# B&R Automation Studio project lab1_MIRTS_save2_4
Automation Studio 4.5.2.102

## Configuration Config1

### Task classes (Cpu.sw)
```
Cyclic#1:
  Program <- Program.prg
Cyclic#4:
  Program1 <- Program1.prg
Binaries: udbdef, TCData, ashwac, arconfig, asfw, ashwd, iomap, User, Role, sysconf
Libraries: MotorCntrl
```

## Configuration labBR

### IoMap.iom - 4PP065_0571_P74/IoMap.iom
```iecst
VAR_CONFIG
	::DoorCtrl:DoorBlock.sw1 AT %IX."X20DI9371".DigitalInput03;
	::DoorCtrl:DoorBlock.sw2 AT %IX."X20DI9371".DigitalInput04;
	::DoorCtrl:DoorBlock.sw3 AT %IX."X20DI9371".DigitalInput05;
	::DoorCtrl:CMD AT %QW."8I64xxxxxxx.00x-1".CMDD_Output;
	::DoorCtrl:ETAD AT %IW."8I64xxxxxxx.00x-1".ETAD_Input;
	::DoorCtrl:Speed AT %QW."8I64xxxxxxx.00x-1".LFRD_Output;
	::LedCtrl:sc0 AT %QX."X20DO9322".DigitalOutput02;
	::LedCtrl:sc1 AT %QX."X20DO9322".DigitalOutput03;
	::LedCtrl:sc2 AT %QX."X20DO9322".DigitalOutput04;
	::LedCtrl:sc3  AT %QX."X20DO9322".DigitalOutput05;
	::DoorCtrl:DoorBlock.sw0 AT %IX."X20DI9371".DigitalInput02;
	::DoorCtrl:DoorBlock.direction AT %IX."X20DI9371".DigitalInput01;
END_VAR
```

### Acp10map.ncm - 4PP065_0571_P74/Motion/Acp10map.ncm
```
NcMapping (NcSwId=Acp10)
  NcObject gAxis01 (ModuleId=X20SM1436, ModuleAddress=SDC_IF1.ST1, Type=ncAXIS, Channel=1, AcoposSimulation=Off, InitParameter=gAxis01i, AcoposParameter=gAxis01a, AdditionalData=CNC_Enabled="1" , Disabled=FALSE, ModuleDisabled=FALSE)
  NcObject gAxis02 (ModuleId=X20SM1436a, ModuleAddress=SDC_IF1.ST2, Type=ncAXIS, Channel=1, AcoposSimulation=Off, InitParameter=gAxis02i, AcoposParameter=gAxis02a, Disabled=FALSE, ModuleDisabled=FALSE)
  NcObject gAxis03 (ModuleId=8I64xxxxxxx.00x-1, ModuleAddress=SDC_IF1.ST3, Type=ncAXIS, Channel=1, AcoposSimulation=Off, InitParameter=gAxis03i, AcoposParameter=gAxis03a, AdditionalData=CNC_Enabled="1" , Disabled=FALSE, ModuleDisabled=FALSE)
  NcObject gAxis04 (ModuleId=X20SM1436b, ModuleAddress=SDC_IF1.ST4, Type=ncAXIS, Channel=1, AcoposSimulation=Off, InitParameter=gAxis04i, AcoposParameter=gAxis04a, AdditionalData=CNC_Enabled="1" , Disabled=FALSE, ModuleDisabled=FALSE)
  NcObject gAxis05 (ModuleId=X20SM1436c, ModuleAddress=SDC_IF1.ST5, Type=ncAXIS, Channel=1, AcoposSimulation=Off, InitParameter=gAxis05i, AcoposParameter=gAxis05a, Disabled=FALSE, ModuleDisabled=FALSE)
```

## Logical view

Binary libraries used (declarations not repeated): Runtime, Operator, AsIecCon, astime, sys_lib, asstring

### Global.var - Global variables
```iecst
VAR
	sw1 : BOOL := FALSE;
	sw2 : BOOL := FALSE;
	sw3 : BOOL := FALSE;
	sw0 : BOOL := FALSE;
END_VAR
```

### Package Logical/Libraries - Global libraries

- Library Logical/Libraries/X64Lib (ANSIC) (no source held here)

### Library Logical/Libraries/GateCtrl (ANSIC)

#### Types.typ
```iecst
TYPE
	GateState :
		(
		ST_INIT := 0,
		ST_UNKNOWN := 1,
		ST_OPEN := 2,
		ST_CLOSE := 3,
		ST_ACC_POS := 4,
		ST_ACC_NEG := 5,
		ST_POS := 6,
		ST_NEG := 7,
		ST_DEC_POS := 8,
		ST_DEC_NEG := 9
		);
END_TYPE
```

#### GateCtrl.fun
```iecst
FUNCTION_BLOCK FBLed
	VAR_OUTPUT
		s1 : BOOL;
		s2 : BOOL;
		s3 : BOOL;
		s4 : BOOL;
	END_VAR
	VAR_INPUT
		State : {REDUND_UNREPLICABLE} GateState;
	END_VAR
END_FUNCTION_BLOCK

{REDUND_ERROR} FUNCTION_BLOCK FBGate (* *) (*$GROUP=User,$CAT=User,$GROUPICON=User.png,$CATICON=User.png*)
	VAR_INPUT
		sw0 : BOOL; (*инпут датчиков*)
		sw1 : BOOL;
		sw2 : BOOL;
		sw3 : BOOL;
		State : {REDUND_UNREPLICABLE} GateState;
		direction : BOOL;
	END_VAR
	VAR_OUTPUT
		Speed : INT;
	END_VAR
	VAR
		DriveBlk : FBX64Inverter;
	END_VAR
END_FUNCTION_BLOCK
```

#### FBGate.c
```c
#include <bur/plctypes.h>
#ifdef __cplusplus
	extern "C"
	{
#endif
	#include "GateCtrl.h"
#ifdef __cplusplus
	};
#endif
/* TODO: Add your comment here */
void FBGate(struct FBGate* inst)
{
	switch (inst->State) {
		case ST_INIT: //
			inst->State = ST_UNKNOWN;
			break;
		case ST_UNKNOWN: //
			if ((inst->direction == 0) && (inst->sw0 == 0)){
			inst->State = ST_OPEN;
			}
			if ((inst->direction == 1) && (inst->sw0 == 1)){
				inst->State = ST_CLOSE;
			}
			break;
		case ST_OPEN: //
			inst->DriveBlk.enable = 0;
			FBX64Inverter(&inst->DriveBlk);
			inst->Speed = 0;
			FBX64Inverter(&inst->DriveBlk);
			if (inst->direction == 1){
				inst->State = ST_ACC_POS;
			}
			break;
		case ST_CLOSE:
			inst->DriveBlk.enable = 0;
			FBX64Inverter(&inst->DriveBlk);
			inst->Speed = 0;
			FBX64Inverter(&inst->DriveBlk);
			if (inst->direction == 0){
				inst->State = ST_ACC_NEG;
			}
			break;
		case ST_ACC_POS:
			inst->DriveBlk.enable = 1;
			inst->Speed = 100;
			FBX64Inverter(&inst->DriveBlk);
			if (inst->sw1){
				inst->State = ST_POS;
			}
			if (inst->direction == 0) {
				inst->State = ST_ACC_NEG;
			}
			break;
		case ST_ACC_NEG:
			inst->DriveBlk.enable = 1;
			FBX64Inverter(&inst->DriveBlk);
			inst->Speed = -100;
			if (!inst->sw2){
				inst->State = ST_NEG;
			}
			break;
		case ST_NEG:
			inst->Speed = -300;
			FBX64Inverter(&inst->DriveBlk);
			if (!inst->sw1){
				inst->State = ST_DEC_NEG;
			}
			break;
		case ST_DEC_NEG:
			inst->Speed = -100;
			FBX64Inverter(&inst->DriveBlk);
			if (!inst->sw0){
				inst->State = ST_OPEN;
			}
			break;
		case ST_DEC_POS:
			FBX64Inverter(&inst->DriveBlk);
			inst->Speed = 100;
			if (inst->sw3){
				inst->State = ST_CLOSE;
			}
			break;
		case ST_POS:
			FBX64Inverter(&inst->DriveBlk);
			inst->Speed = 300;
			if (inst->sw2){
				inst->State = ST_DEC_POS;
			}
			if (inst->direction == 0) {
				inst->State = ST_NEG;
			}
			break;
	}
}
```

### arnc0man.typ
```iecst
TYPE
ARNC0SWVER_typ : STRUCT                                     (* Software Version ID *)
   NOT_USE_1            : ARRAY [0..1] OF USINT ;
   nc_system_device     : UINT ;                            (* ACOPOS operating system *)
   nc_manager           : UINT ;                            (* NC manager *)
   nc_system            : UINT ;                            (* NC operating system *)
END_STRUCT;
ARNC0OBIHW_typ : STRUCT                                     (* Hardware information *)
   init                 : USINT ;                           (* Initialized *)
   reserve1             : USINT ;                           (* Reserved *)
   acp_id               : USINT ;                           (* ACOPOS ID *)
   acp_id_nr            : USINT ;                           (* ACOPOS ID production number *)
   acp_typ              : USINT ;                           (* ACOPOS type *)
   ax_num               : USINT ;                           (* Number of axes (power stages) *)
   reserve2             : UINT ;                            (* Reserved *)
   product_code         : UDINT ;                           (* Product code *)
   serial_nr            : UDINT ;                           (* Serial number *)
END_STRUCT;
ARNC0OBINF_typ : STRUCT                                     (* NC Object Information *)
   net_if_typ           : UINT ;                            (* Network interface type *)
   net_if_idx           : UINT ;                            (* Network interface index *)
   node_nr              : UINT ;                            (* Drive node number *)
   nc_obj_typ           : UINT ;                            (* NC object type *)
   nc_obj_idx           : UINT ;                            (* NC object index *)
   reserve              : UINT ;                            (* Reserved *)
   nc_obj_name          : ARRAY [0..47] OF USINT ;          (* NC object name *)
   hardware             : ARNC0OBIHW_typ ;                  (* Hardware information *)
END_STRUCT;
ARNC0AXSIM_typ : STRUCT                                     (* Simulation mode *)
   NOT_USE_1            : ARRAY [0..3] OF USINT ;
   status               : UINT ;                            (* Status *)
   mode                 : UINT ;                            (* Mode *)
   NOT_USE_2            : ARRAY [0..47] OF USINT ;
END_STRUCT;
ARNC0GLIPA_typ : STRUCT                                     (* INIT Parameters *)
   ok                   : USINT ;                           (* Operation complete *)
   error                : USINT ;                           (* Error *)
   reserve              : UINT ;                            (* Reserved *)
   datobj_ident         : UDINT ;                           (* Data object ident *)
   data_modul           : ARRAY [0..11] OF USINT ;          (* Name of the data module *)
END_STRUCT;
ARNC0GLINI_typ : STRUCT                                     (* Global Initialization *)
   init                 : USINT ;                           (* Global Initialization complete *)
   NOT_USE_1            : ARRAY [0..2] OF USINT ;
   init_par             : ARNC0GLIPA_typ ;                  (* INIT Parameters *)
END_STRUCT;
ARNC0NSVRQ_typ : STRUCT                                     (* Request (to the drive) *)
   par_id               : UINT ;                            (* Parameter ID *)
   NOT_USE_1            : ARRAY [0..1] OF USINT ;
END_STRUCT;
ARNC0NSVRS_typ : STRUCT                                     (* Response (from the drive) *)
   par_id               : UINT ;                            (* Parameter ID *)
   NOT_USE_1            : ARRAY [0..1] OF USINT ;
END_STRUCT;
ARNC0NETSV_typ : STRUCT                                     (* Service Interface *)
   data_adr             : UDINT ;                           (* Data address *)
   data_text            : ARRAY [0..31] OF USINT ;          (* Data in text format *)
   request              : ARNC0NSVRQ_typ ;                  (* Request (to the drive) *)
   response             : ARNC0NSVRS_typ ;                  (* Response (from the drive) *)
END_STRUCT;
ARNC0NETAX_typ : STRUCT                                     (* Network *)
   init                 : USINT ;                           (* Network initialized *)
   phase                : USINT ;                           (* Phase *)
   NOT_USE_1            : USINT ;
   nc_sys_restart       : USINT ;                           (* A Restart of the NC operating system was executed *)
   reserve              : UINT ;                            (* Reserved *)
   reserve1             : UINT ;                            (* Reserved *)
   service              : ARNC0NETSV_typ ;                  (* Service Interface *)
END_STRUCT;
ARNC0AXDBS_typ : STRUCT                                     (* Status *)
   ok                   : USINT ;                           (* Operation complete *)
   error                : USINT ;                           (* Error *)
   reserve1             : USINT ;                           (* Reserved *)
   reserve2             : USINT ;                           (* Reserved *)
   data_len             : UDINT ;                           (* Length of data *)
   datobj_ident         : UDINT ;                           (* Data object ident *)
   datobj_datadr        : UDINT ;                           (* Address of the data object data *)
END_STRUCT;
ARNC0AXDBP_typ : STRUCT                                     (* Parameters *)
   file_device          : ARRAY [0..31] OF USINT ;          (* Name of File Device *)
   datobj_name          : ARRAY [0..31] OF USINT ;          (* Name of the data object *)
   datobj_type          : UINT ;                            (* Type of the data object *)
   datblock_par_id      : UINT ;                            (* Parameter ID of the data block *)
   idx1_par_id          : UINT ;                            (* Parameter ID of data block index 1 *)
   idx1                 : UINT ;                            (* Data block index 1 *)
   idx2_par_id          : UINT ;                            (* Parameter ID of data block index 2 *)
   idx2                 : UINT ;                            (* Data block index 2 *)
   NOT_USE_1            : ARRAY [0..7] OF USINT ;
END_STRUCT;
ARNC0AXDBL_typ : STRUCT                                     (* Data block operation *)
   status               : ARNC0AXDBS_typ ;                  (* Status *)
   parameter            : ARNC0AXDBP_typ ;                  (* Parameters *)
END_STRUCT;
ARNC0DISTA_typ : STRUCT                                     (* Status *)
   reference            : USINT ;                           (* Reference switch *)
   pos_hw_end           : USINT ;                           (* Positive HW end switch *)
   neg_hw_end           : USINT ;                           (* Negative HW end switch *)
   trigger1             : USINT ;                           (* Trigger1 *)
   trigger2             : USINT ;                           (* Trigger2 *)
   enable               : USINT ;                           (* Enable *)
   NOT_USE_1            : ARRAY [0..1] OF USINT ;
END_STRUCT;
ARNC0DILEV_typ : STRUCT                                     (* Active Input Level *)
   reference            : UINT ;                            (* Reference switch *)
   pos_hw_end           : UINT ;                            (* Positive HW end switch *)
   neg_hw_end           : UINT ;                            (* Negative HW end switch *)
   trigger1             : UINT ;                            (* Trigger1 *)
   trigger2             : UINT ;                            (* Trigger2 *)
   NOT_USE_1            : ARRAY [0..1] OF USINT ;
END_STRUCT;
ARNC0DIFRC_typ : STRUCT                                     (* Set status of digital inputs via force function *)
   reference            : USINT ;                           (* Reference switch *)
   pos_hw_end           : USINT ;                           (* Positive HW end switch *)
   neg_hw_end           : USINT ;                           (* Negative HW end switch *)
   trigger1             : USINT ;                           (* Trigger1 *)
   trigger2             : USINT ;                           (* Trigger2 *)
   reserve1             : USINT ;                           (* Reserved *)
   reserve2             : UINT ;                            (* Reserved *)
END_STRUCT;
ARNC0DIGIN_typ : STRUCT                                     (* Digital Inputs *)
   init                 : USINT ;                           (* Digital inputs initialized *)
   NOT_USE_1            : ARRAY [0..2] OF USINT ;
   status               : ARNC0DISTA_typ ;                  (* Status *)
   level                : ARNC0DILEV_typ ;                  (* Active Input Level *)
   force                : ARNC0DIFRC_typ ;                  (* Set status of digital inputs via force function *)
END_STRUCT;
ARNC0ENCSL_typ : STRUCT                                     (* Load *)
   units                : UDINT ;                           (* Units at the load *)
   rev_motor            : UDINT ;                           (* Motor revolutions *)
END_STRUCT;
ARNC0ENCSC_typ : STRUCT                                     (* Scale of encoder interface *)
   load                 : ARNC0ENCSL_typ ;                  (* Load *)
END_STRUCT;
ARNC0ENCPA_typ : STRUCT                                     (* Parameters of encoder interface *)
   count_dir            : USINT ;                           (* Count direction *)
   NOT_USE_1            : ARRAY [0..2] OF USINT ;
   scaling              : ARNC0ENCSC_typ ;                  (* Scaling *)
END_STRUCT;
ARNC0ENCIF_typ : STRUCT                                     (* Encoder interface *)
   init                 : USINT ;                           (* Encoder interface initialized *)
   NOT_USE_1            : ARRAY [0..2] OF USINT ;
   parameter            : ARNC0ENCPA_typ ;                  (* Parameters *)
END_STRUCT;
ARNC0AXLPA_typ : STRUCT                                     (* Parameters *)
   v_pos                : REAL ;                            (* Speed in positive direction *)
   v_neg                : REAL ;                            (* Speed in negative direction *)
   a1_pos               : REAL ;                            (* Acceleration in positive direction *)
   a2_pos               : REAL ;                            (* Deceleration in positive direction *)
   a1_neg               : REAL ;                            (* Acceleration in negative direction *)
   a2_neg               : REAL ;                            (* Deceleration in negative direction *)
   t_jolt               : REAL ;                            (* Jolt time *)
   t_in_pos             : REAL ;                            (* Settling time before message "In Position" *)
   pos_sw_end           : DINT ;                            (* Positive SW end *)
   neg_sw_end           : DINT ;                            (* Negative SW end *)
   sw_end_enable        : USINT ;                           (* Control byte for limit monitor *)
   sl_chain             : USINT ;                           (* Slaves in a chain or ncOFF *)
   NOT_USE_1            : ARRAY [0..1] OF USINT ;
   ds_warning           : REAL ;                            (* Lag error limit for display of a warning *)
   ds_stop              : REAL ;                            (* Lag error limit for stop of a movement *)
   a_stop               : REAL ;                            (* Acceleration limit for stop of a movement *)
   dv_stop              : REAL ;                            (* Speed error limit for stop of a movement *)
   dv_stop_mode         : UDINT ;                           (* Mode for speed error monitoring *)
END_STRUCT;
ARNC0AXLIM_typ : STRUCT                                     (* Limit values *)
   init                 : USINT ;                           (* Axis limit values initialized *)
   status               : USINT ;                           (* Status *)
   NOT_USE_1            : ARRAY [0..1] OF USINT ;
   parameter            : ARNC0AXLPA_typ ;                  (* Parameters *)
END_STRUCT;
ARNC0CTRPO_typ : STRUCT                                     (* Position controller *)
   kv                   : REAL ;                            (* Proportional amplification *)
   tn                   : REAL ;                            (* Integral action time *)
   t_predict            : REAL ;                            (* Prediction time *)
   t_total              : REAL ;                            (* Total time *)
   p_max                : REAL ;                            (* Maximum proportional action *)
   i_max                : REAL ;                            (* Maximum integral action *)
END_STRUCT;
ARNC0ISQFI_typ : STRUCT                                     (* ISQ Filter *)
   type                 : UINT ;                            (* Type *)
   reserve              : UINT ;                            (* Reserved *)
   a0                   : REAL ;                            (* Coefficient a0 *)
   a1                   : REAL ;                            (* Coefficient a1 *)
   b0                   : REAL ;                            (* Coefficient b0 *)
   b1                   : REAL ;                            (* Coefficient b1 *)
   b2                   : REAL ;                            (* Coefficient b2 *)
   c0_par_id            : UINT ;                            (* Parameter ID for coefficient c0 *)
   c1_par_id            : UINT ;                            (* Parameter ID for coefficient c1 *)
END_STRUCT;
ARNC0CTRSP_typ : STRUCT                                     (* Speed controller *)
   kv                   : REAL ;                            (* Proportional amplification *)
   tn                   : REAL ;                            (* Integral action time *)
   t_filter             : REAL ;                            (* Filter time constant *)
   isq_filter1          : ARNC0ISQFI_typ ;                  (* ISQ Filter1 *)
   isq_filter2          : ARNC0ISQFI_typ ;                  (* ISQ Filter2 *)
   isq_filter3          : ARNC0ISQFI_typ ;                  (* ISQ Filter3 *)
END_STRUCT;
ARNC0CTRUF_typ : STRUCT                                     (* U/f Control *)
   type                 : USINT ;                           (* Type *)
   auto_config          : USINT ;                           (* Automatic configuration *)
   reserve              : UINT ;                            (* Reserved *)
   u0                   : REAL ;                            (* Boost voltage *)
   un                   : REAL ;                            (* Rated voltage *)
   fn                   : REAL ;                            (* Rated frequency *)
   k_f_slip             : REAL ;                            (* Slip compensation: Multiplication factor of compensated frequency *)
END_STRUCT;
ARNC0CTRFF_typ : STRUCT                                     (* Feed Forward Control *)
   torque_load          : REAL ;                            (* Load torque *)
   torque_pos           : REAL ;                            (* Torque in positive direction *)
   torque_neg           : REAL ;                            (* Torque in negative direction *)
   kv_torque            : REAL ;                            (* Speed torque factor *)
   inertia              : REAL ;                            (* Mass moment of inertia *)
   t_filter_a           : REAL ;                            (* Acceleration filter time constant *)
END_STRUCT;
ARNC0CTRL_typ : STRUCT                                      (* Controller *)
   init                 : USINT ;                           (* Controller initialized *)
   ready                : USINT ;                           (* Ready *)
   status               : USINT ;                           (* Status *)
   mode                 : USINT ;                           (* Mode *)
   position             : ARNC0CTRPO_typ ;                  (* Position Controller *)
   speed                : ARNC0CTRSP_typ ;                  (* Speed Controller *)
   uf                   : ARNC0CTRUF_typ ;                  (* U/f Control *)
   ff                   : ARNC0CTRFF_typ ;                  (* Feed Forward Control *)
END_STRUCT;
ARNC0AXSTI_typ : STRUCT                                     (* Index of Parameter Record *)
   command              : USINT ;                           (* for the next stop command *)
   NOT_USE_1            : ARRAY [0..2] OF USINT ;
END_STRUCT;
ARNC0AXSTP_typ : STRUCT                                     (* Parameter Records *)
   decel_ramp           : USINT ;                           (* Deceleration ramp *)
   controller           : USINT ;                           (* Controller state after movement abortion *)
   NOT_USE_1            : ARRAY [0..1] OF USINT ;
END_STRUCT;
ARNC0AXSTQ_typ : STRUCT                                     (* Quickstop *)
   decel_ramp           : USINT ;                           (* Deceleration ramp *)
   NOT_USE_1            : USINT ;
   reserve2             : UINT ;                            (* Reserved *)
   NOT_USE_2            : ARRAY [0..3] OF USINT ;
END_STRUCT;
ARNC0AXSTD_typ : STRUCT                                     (* Drive error *)
   decel_ramp           : USINT ;                           (* Deceleration ramp *)
   reserve1             : USINT ;                           (* Reserved *)
   reserve2             : UINT ;                            (* Reserved *)
END_STRUCT;
ARNC0AXSTO_typ : STRUCT                                     (* Stop Movement *)
   init                 : USINT ;                           (* Stop initialized *)
   NOT_USE_1            : ARRAY [0..2] OF USINT ;
   index                : ARNC0AXSTI_typ ;                  (* Index *)
   parameter            : ARRAY [0..3] OF ARNC0AXSTP_typ ;  (* Parameter record *)
   quickstop            : ARNC0AXSTQ_typ ;                  (* Quickstop *)
   drive_error          : ARNC0AXSTD_typ ;                  (* Drive error *)
END_STRUCT;
ARNC0HOMST_typ : STRUCT                                     (* Status *)
   ok                   : USINT ;                           (* Reference position valid *)
   NOT_USE_1            : ARRAY [0..2] OF USINT ;
   tr_s_rel             : REAL ;                            (* Distance between activation of "triggering reference pulse" and the occurrence of the reference pulse *)
   offset               : DINT ;                            (* Home offset after completion of homing procedure *)
END_STRUCT;
ARNC0HOMPA_typ : STRUCT                                     (* Parameters *)
   s                    : DINT ;                            (* Reference position *)
   v_switch             : REAL ;                            (* Speed for searching the reference switch *)
   v_trigger            : REAL ;                            (* Trigger speed (after ref. switch has been reached) *)
   a                    : REAL ;                            (* Acceleration *)
   mode                 : USINT ;                           (* Mode *)
   edge                 : USINT ;                           (* Edge of reference switch *)
   start_dir            : USINT ;                           (* Start direction *)
   trigg_dir            : USINT ;                           (* Trigger direction *)
   ref_pulse            : USINT ;                           (* Reference pulse *)
   fix_dir              : USINT ;                           (* Fixed direction *)
   reserve1             : USINT ;                           (* Reserved *)
   reserve2             : USINT ;                           (* Reserved *)
   tr_s_block           : REAL ;                            (* Reference pulse block distance *)
   torque_lim           : REAL ;                            (* Torque limit for homing on block *)
   ds_block             : REAL ;                            (* Lag error for block detection *)
   ds_stop              : REAL ;                            (* Lag error for stop of a movement *)
END_STRUCT;
ARNC0HOME_typ : STRUCT                                      (* Homing *)
   init                 : USINT ;                           (* Homing procedure initialized *)
   NOT_USE_1            : ARRAY [0..2] OF USINT ;
   status               : ARNC0HOMST_typ ;                  (* Status *)
   parameter            : ARNC0HOMPA_typ ;                  (* Parameters *)
END_STRUCT;
ARNC0BMVST_typ : STRUCT                                     (* Status *)
   in_pos               : USINT ;                           (* "In Position" (target position reached) *)
   reserve              : ARRAY [0..2] OF USINT ;           (* Reserved *)
END_STRUCT;
ARNC0BMVOV_typ : STRUCT                                     (* Override *)
   v                    : UINT ;                            (* Speed override *)
   NOT_USE_1            : ARRAY [0..1] OF USINT ;
END_STRUCT;
ARNC0BMVPA_typ : STRUCT                                     (* Parameters *)
   s                    : DINT ;                            (* Target position or relative move distance *)
   v_pos                : REAL ;                            (* Speed in positive direction *)
   v_neg                : REAL ;                            (* Speed in negative direction *)
   a1_pos               : REAL ;                            (* Acceleration in positive direction *)
   a2_pos               : REAL ;                            (* Deceleration in positive direction *)
   a1_neg               : REAL ;                            (* Acceleration in negative direction *)
   a2_neg               : REAL ;                            (* Deceleration in negative direction *)
END_STRUCT;
ARNC0TRG_typ : STRUCT                                       (* Source for Hardware Trigger *)
   nc_object            : UDINT ;                           (* NC object or ncOFF *)
   NOT_USE_1            : ARRAY [0..7] OF USINT ;
END_STRUCT;
ARNC0TRSTP_typ : STRUCT                                     (* Mode "Stop after trigger" *)
   init                 : USINT ;                           (* Initialized *)
   event                : USINT ;                           (* Event *)
   NOT_USE_1            : ARRAY [0..1] OF USINT ;
   s_rest               : DINT ;                            (* Remaining distance after trigger *)
   trg_source           : ARNC0TRG_typ ;                    (* Trigger Source *)
END_STRUCT;
ARNC0BAMOV_typ : STRUCT                                     (* Basis Movements *)
   init                 : USINT ;                           (* Initialized *)
   reserve0             : ARRAY [0..2] OF USINT ;           (* Reserved *)
   status               : ARNC0BMVST_typ ;                  (* Status *)
   override             : ARNC0BMVOV_typ ;                  (* Override *)
   parameter            : ARNC0BMVPA_typ ;                  (* Parameters *)
   trg_stop             : ARNC0TRSTP_typ ;                  (* Mode "Stop after trigger" *)
END_STRUCT;
ARNC0AXMOV_typ : STRUCT                                     (* Axis Movement *)
   mode                 : UINT ;                            (* Mode *)
   detail               : UINT ;                            (* Detail *)
   stop                 : ARNC0AXSTO_typ ;                  (* Stop Movement *)
   homing               : ARNC0HOME_typ ;                   (* Homing procedure *)
   basis                : ARNC0BAMOV_typ ;                  (* Basis movements *)
END_STRUCT;
ARNC0SUOST_typ : STRUCT                                     (* Status *)
   ident                : UDINT ;                           (* Ident of data object *)
   ok                   : USINT ;                           (* Operation complete *)
   error                : USINT ;                           (* Error *)
   reserve1             : USINT ;                           (* Reserved *)
   reserve2             : USINT ;                           (* Reserved *)
END_STRUCT;
ARNC0SUOPA_typ : STRUCT                                     (* Parameters *)
   name                 : ARRAY [0..11] OF USINT ;          (* Name of data object *)
END_STRUCT;
ARNC0SUOBJ_typ : STRUCT                                     (* Data object *)
   status               : ARNC0SUOST_typ ;                  (* Status *)
   parameter            : ARNC0SUOPA_typ ;                  (* Parameters *)
END_STRUCT;
ARNC0SUMAS_typ : STRUCT                                     (* Status *)
   mode                 : UINT ;                            (* Mode *)
   ok                   : USINT ;                           (* Operation complete *)
   error                : USINT ;                           (* Error *)
   quality              : REAL ;                            (* Quality of parameter identification *)
END_STRUCT;
ARNC0SUMAO_typ : STRUCT                                     (* Optional parameters *)
   z_p                  : USINT ;                           (* Number of polepairs *)
   phase                : USINT ;                           (* Phase *)
   reserve2             : UINT ;                            (* Reserved *)
   u_const              : REAL ;                            (* Voltage constant *)
   v_max                : REAL ;                            (* Maximum speed *)
   trq_0                : REAL ;                            (* Stall  torque *)
   trq_n                : REAL ;                            (* Rated torque *)
   trq_max              : REAL ;                            (* Peak  torque *)
   trq_const            : REAL ;                            (* Torque constant *)
   i_0                  : REAL ;                            (* Stall current *)
   i_max                : REAL ;                            (* Peak current *)
   i_m                  : REAL ;                            (* Magnetizing current *)
   phase_cross_sect     : REAL ;                            (* Cross section of a phase *)
   invcl_a1             : REAL ;                            (* Inverter characteristic: Gain factor *)
   invcl_a2             : REAL ;                            (* Inverter characteristic: Exponent *)
END_STRUCT;
ARNC0SUMAP_typ : STRUCT                                     (* Parameters *)
   mode                 : UINT ;                            (* Mode *)
   reserve              : UINT ;                            (* Reserved *)
   u_n                  : REAL ;                            (* Rated voltage *)
   i_n                  : REAL ;                            (* Rated current *)
   v_n                  : REAL ;                            (* Rated speed *)
   f_n                  : REAL ;                            (* Rated frequency *)
   cos_phi              : REAL ;                            (* Active power factor *)
   t_tripping_therm     : REAL ;                            (* Tripping time at thermal overload *)
   optional             : ARNC0SUMAO_typ ;                  (* Optional parameters *)
END_STRUCT;
ARNC0SUMA_typ : STRUCT                                      (* Induction motor *)
   status               : ARNC0SUMAS_typ ;                  (* Status *)
   parameter            : ARNC0SUMAP_typ ;                  (* Parameters *)
END_STRUCT;
ARNC0SUMSS_typ : STRUCT                                     (* Status *)
   mode                 : UINT ;                            (* Mode *)
   ok                   : USINT ;                           (* Operation complete *)
   error                : USINT ;                           (* Error *)
   quality              : REAL ;                            (* Quality of parameter identification *)
END_STRUCT;
ARNC0SUMSO_typ : STRUCT                                     (* Optional parameters *)
   phase                : USINT ;                           (* Phase *)
   reserve1             : USINT ;                           (* Reserved *)
   reserve2             : UINT ;                            (* Reserved *)
   u_const              : REAL ;                            (* Voltage constant *)
   v_max                : REAL ;                            (* Maximum speed *)
   trq_0                : REAL ;                            (* Stall  torque *)
   trq_const            : REAL ;                            (* Torque constant *)
   i_0                  : REAL ;                            (* Stall current *)
   phase_cross_sect     : REAL ;                            (* Cross section of a phase *)
   invcl_a1             : REAL ;                            (* Inverter characteristic: Gain factor *)
   invcl_a2             : REAL ;                            (* Inverter characteristic: Exponent *)
END_STRUCT;
ARNC0SUMSP_typ : STRUCT                                     (* Parameters *)
   mode                 : UINT ;                            (* Mode *)
   z_p                  : USINT ;                           (* Number of polepairs *)
   reserve              : USINT ;                           (* Reserved *)
   u_n                  : REAL ;                            (* Rated voltage *)
   i_n                  : REAL ;                            (* Rated current *)
   v_n                  : REAL ;                            (* Rated speed *)
   trq_n                : REAL ;                            (* Rated torque *)
   trq_max              : REAL ;                            (* Peak  torque *)
   i_max                : REAL ;                            (* Peak current *)
   t_tripping_therm     : REAL ;                            (* Tripping time at thermal overload *)
   optional             : ARNC0SUMSO_typ ;                  (* Optional parameters *)
END_STRUCT;
ARNC0SUMS_typ : STRUCT                                      (* Synchronous motor *)
   status               : ARNC0SUMSS_typ ;                  (* Status *)
   parameter            : ARNC0SUMSP_typ ;                  (* Parameters *)
END_STRUCT;
ARNC0SUPHS_typ : STRUCT                                     (* Status *)
   mode                 : UINT ;                            (* Mode *)
   ok                   : USINT ;                           (* Operation complete *)
   error                : USINT ;                           (* Error *)
   rho_0                : REAL ;                            (* Commutation offset *)
   z_p                  : USINT ;                           (* Number of polepairs *)
   reserve1             : USINT ;                           (* Reserved *)
   reserve2             : UINT ;                            (* Reserved *)
END_STRUCT;
ARNC0SUPHP_typ : STRUCT                                     (* Parameters *)
   mode                 : UINT ;                            (* Mode *)
   reserve              : UINT ;                            (* Reserved *)
   i                    : REAL ;                            (* Current *)
   t                    : REAL ;                            (* Time *)
END_STRUCT;
ARNC0SUPH_typ : STRUCT                                      (* Motor phasing *)
   status               : ARNC0SUPHS_typ ;                  (* Status *)
   parameter            : ARNC0SUPHP_typ ;                  (* Parameters *)
END_STRUCT;
ARNC0SUCST_typ : STRUCT                                     (* Status *)
   mode                 : UINT ;                            (* Mode *)
   ok                   : USINT ;                           (* Operation complete *)
   error                : USINT ;                           (* Error *)
END_STRUCT;
ARNC0SUCPA_typ : STRUCT                                     (* Parameters *)
   mode                 : UINT ;                            (* Mode *)
   orientation          : USINT ;                           (* Orientation *)
   operating_point      : USINT ;                           (* Operating point *)
   i_max_percent        : REAL ;                            (* Maximum percentage for rated current *)
   v_max_percent        : REAL ;                            (* Maximum percentage for speed limit value *)
   s_max                : DINT ;                            (* Maximum move distance *)
   ds_max               : REAL ;                            (* Maximum lag error *)
   kv_percent           : REAL ;                            (* Percentage for proportional amplification *)
   signal_order         : UDINT ;                           (* Order of excitation signal *)
   kv_max               : REAL ;                            (* Maximum proportional amplification *)
   a                    : REAL ;                            (* Acceleration *)
   signal_type          : UINT ;                            (* Type of the excitation signal *)
   reserve              : UINT ;                            (* Reserved *)
   signal_f_start       : REAL ;                            (* Start frequency of the excitation signal *)
   signal_f_stop        : REAL ;                            (* Stop frequency of the excitation signal *)
   signal_time          : REAL ;                            (* Duration of the excitation signal *)
END_STRUCT;
ARNC0SUCTR_typ : STRUCT                                     (* Controller *)
   status               : ARNC0SUCST_typ ;                  (* Status *)
   parameter            : ARNC0SUCPA_typ ;                  (* Parameters *)
END_STRUCT;
ARNC0SUIRS_typ : STRUCT                                     (* Status *)
   mode                 : UINT ;                            (* Mode *)
   ok                   : USINT ;                           (* Operation complete *)
   error                : USINT ;                           (* Error *)
   quality              : REAL ;                            (* Quality of parameter identification *)
END_STRUCT;
ARNC0SUIRP_typ : STRUCT                                     (* Parameters *)
   mode                 : UINT ;                            (* Mode *)
   reserve              : USINT ;                           (* Reserved *)
   ref_system           : USINT ;                           (* Reference system *)
   pos_offset           : REAL ;                            (* Position offset *)
   v                    : REAL ;                            (* Speed *)
END_STRUCT;
ARNC0SUIR_typ : STRUCT                                      (* ISQ-Ripple *)
   status               : ARNC0SUIRS_typ ;                  (* Status *)
   parameter            : ARNC0SUIRP_typ ;                  (* Parameters *)
END_STRUCT;
ARNC0SETUP_typ : STRUCT                                     (* Setup *)
   status               : USINT ;                           (* Status *)
   reserve              : USINT ;                           (* Reserved *)
   detail               : UINT ;                            (* Detail *)
   datobj               : ARNC0SUOBJ_typ ;                  (* Data object *)
   motor_induction      : ARNC0SUMA_typ ;                   (* Induction motor *)
   motor_synchron       : ARNC0SUMS_typ ;                   (* Synchronous motor *)
   motor_phasing        : ARNC0SUPH_typ ;                   (* Motor phasing *)
   controller           : ARNC0SUCTR_typ ;                  (* Controller *)
   isq_ripple           : ARNC0SUIR_typ ;                   (* ISQ-Ripple *)
END_STRUCT;
ARNC0PLCOPENAX_typ : STRUCT                                 (* PLCopen *)
   PLCopen_AxState      : USINT ;                           (* PLCopen axis state *)
   NOT_USE_1            : ARRAY [0..2] OF USINT ;
END_STRUCT;
ARNC0ACTST_typ : STRUCT                                     (* Status *)
   active               : USINT ;                           (* Active *)
   complete             : USINT ;                           (* Complete *)
   NOT_USE_1            : ARRAY [0..1] OF USINT ;
END_STRUCT;
ARNC0LATCH_typ : STRUCT                                     (* Position latch *)
   status               : ARNC0ACTST_typ ;                  (* Status *)
   position             : DINT ;                            (* Latchposition *)
   position2            : DINT ;                            (* Second latchposition *)
   event                : USINT ;                           (* Event *)
   reserve              : ARRAY [0..2] OF USINT ;           (* Reserved *)
   window               : DINT ;                            (* Latch window *)
   w_position           : DINT ;                            (* Position of the latch window *)
END_STRUCT;
ARNC0POS_L_typ : STRUCT                                     (* Position latches *)
   latch1               : ARNC0LATCH_typ ;                  (* Positioning latch 1 *)
   latch2               : ARNC0LATCH_typ ;                  (* Positioning latch 2 *)
END_STRUCT;
ARNC0CPRST_typ : STRUCT                                     (* Status *)
   active               : USINT ;                           (* Active *)
   index                : USINT ;                           (* Index *)
   cnt_start            : USINT ;                           (* Number of not acknowledged start commands *)
   reserve              : USINT ;                           (* Reserved *)
   curr_prof            : ARRAY [0..11] OF USINT ;          (* Name of current cam profile *)
END_STRUCT;
ARNC0CPRPA_typ : STRUCT                                     (* Parameters *)
   mode                 : USINT ;                           (* Mode *)
   reserve0             : ARRAY [0..2] OF USINT ;           (* Reserved *)
   ma_ax                : UDINT ;                           (* NC object of the master axis *)
   ma_add_ax            : UDINT ;                           (* NC object of the additive axis of the master axis *)
   sl_add_ax            : UDINT ;                           (* NC object of the additive axis of the slave  axis *)
   ma_s_start           : DINT ;                            (* Start position of the master axis *)
   ma_ivstart           : UDINT ;                           (* Start interval of the master axis *)
   ma_add_el            : REAL ;                            (* "Additive" element of the master axis *)
   ma_factor            : REAL ;                            (* Multiplication factor for the master axis *)
   ma_add_fa            : REAL ;                            (* Multiplication factor for the "additive" axis of the master axis *)
   sl_add_el            : REAL ;                            (* "Additive" element of the slave axis *)
   sl_factor            : REAL ;                            (* Multiplication factor for the slave  axis *)
   sl_add_fa            : REAL ;                            (* Multiplication factor for the "additive" axis of the slave axis *)
   factor_set           : USINT ;                           (* Set multiplication factors "ma/sl_factor" *)
   reserve              : ARRAY [0..2] OF USINT ;           (* Reserved *)
   reserve1             : ARRAY [0..5] OF UDINT ;           (* Reserved *)
END_STRUCT;
ARNC0CPRDM_typ : STRUCT                                     (* Data Modules *)
   single               : ARRAY [0..11] OF USINT ;          (* Name of the entry cam profile *)
   cyclic               : ARRAY [0..11] OF USINT ;          (* Name of the cyclic cam profile *)
END_STRUCT;
ARNC0CPINF_typ : STRUCT                                     (* INFO Function *)
   status               : ARNC0ACTST_typ ;                  (* Status *)
   sl_s_rel             : DINT ;                            (* Relative position of slave axis in the cam profile *)
   ma_s_rel             : UDINT ;                           (* Relative position of master axis in the cam profile *)
END_STRUCT;
ARNC0CPRCG_typ : STRUCT                                     (* Compensation Gears *)
   ma_v_max             : REAL ;                            (* Maximum speed of the master axis *)
   ma_s_comp            : DINT ;                            (* Compensation distance of master axis *)
   sl_s_comp            : DINT ;                            (* Compensation distance of slave axis *)
END_STRUCT;
ARNC0CAMPR_typ : STRUCT                                     (* Electronic Cam Profile *)
   status               : ARNC0CPRST_typ ;                  (* Status *)
   parameter            : ARNC0CPRPA_typ ;                  (* Parameters *)
   data_modul           : ARNC0CPRDM_typ ;                  (* Data Modules *)
   info                 : ARNC0CPINF_typ ;                  (* INFO-function *)
   co_gears             : ARNC0CPRCG_typ ;                  (* Compensation gear *)
END_STRUCT;
ARNC0AUTSP_typ : STRUCT                                     (* Parameters *)
   index                : USINT ;                           (* Index *)
   reserve              : ARRAY [0..2] OF USINT ;           (* Reserved *)
END_STRUCT;
ARNC0AUTST_typ : STRUCT                                     (* Status *)
   init                 : USINT ;                           (* Initialized *)
   active               : USINT ;                           (* Active *)
   st_type              : USINT ;                           (* Type of the actual state *)
   st_index             : USINT ;                           (* Index of the actual state *)
   cam_prof             : ARNC0AUTSP_typ ;                  (* Cam profile *)
END_STRUCT;
ARNC0AUTID_typ : STRUCT                                     (* INIT State *)
   st_type              : USINT ;                           (* Type of the state to initialize *)
   st_index             : USINT ;                           (* Type of the state to initialize *)
   NOT_USE_1            : ARRAY [0..1] OF USINT ;
END_STRUCT;
ARNC0AUTCC_typ : STRUCT                                     (* Coupling Configuration *)
   ma_ax                : UDINT ;                           (* NC object of the master axis *)
   ma_add_ax            : UDINT ;                           (* NC object of the additive axis of the master axis *)
   sl_add_ax            : UDINT ;                           (* NC object of the additive axis of the slave  axis *)
END_STRUCT;
ARNC0AUTGL_typ : STRUCT                                     (* Global Parameters *)
   ma_add_el            : REAL ;                            (* "Additive" element of the master axis *)
   sl_add_el            : REAL ;                            (* "Additive" element of the slave axis *)
END_STRUCT;
ARNC0AUTEB_typ : STRUCT                                     (* Events for basis state *)
   type                 : USINT ;                           (* Type *)
   NOT_USE_1            : ARRAY [0..2] OF USINT ;
   trg_source           : ARNC0TRG_typ ;                    (* Trigger Source *)
   attribute            : USINT ;                           (* Attribute *)
   st_type              : USINT ;                           (* Type of the next state *)
   st_index             : USINT ;                           (* Index  of the next state *)
   NOT_USE_2            : USINT ;
END_STRUCT;
ARNC0AUTBA_typ : STRUCT                                     (* Basis State *)
   ma_s_start           : DINT ;                            (* Start position of the master axis *)
   ma_ivstart           : UDINT ;                           (* Start interval of the master axis *)
   event                : ARRAY [0..5] OF ARNC0AUTEB_typ ;  (* Event *)
END_STRUCT;
ARNC0AUTCG_typ : STRUCT                                     (* Compensation Gears *)
   ma_v_max             : REAL ;                            (* Maximum speed of the master axis *)
   ma_s_rel             : DINT ;                            (* Relative distance of the master axis *)
   sl_s_rel             : DINT ;                            (* Relative distance of the slave axis *)
   ma_s_min             : DINT ;                            (* Minimum distance of the master axis *)
   mode                 : USINT ;                           (* Mode *)
   reserve              : ARRAY [0..2] OF USINT ;           (* Reserved *)
END_STRUCT;
ARNC0AUTCP_typ : STRUCT                                     (* Cam Profile *)
   name                 : ARRAY [0..11] OF USINT ;          (* Name of the NC data module *)
   ma_factor            : REAL ;                            (* Multiplication factor for the master axis *)
   sl_factor            : REAL ;                            (* Multiplication factor for the slave  axis *)
END_STRUCT;
ARNC0AUTER_typ : STRUCT                                     (* Events for automat states *)
   type                 : USINT ;                           (* Type *)
   NOT_USE_1            : ARRAY [0..2] OF USINT ;
   trg_source           : ARNC0TRG_typ ;                    (* Trigger Source *)
   attribute            : USINT ;                           (* Attribute *)
   st_type              : USINT ;                           (* Type of the next state *)
   st_index             : USINT ;                           (* Index  of the next state *)
   NOT_USE_2            : USINT ;
END_STRUCT;
ARNC0AUTSC_typ : STRUCT                                     (* States *)
   count                : UINT ;                            (* Count *)
   NOT_USE_1            : ARRAY [0..1] OF USINT ;
   co_gears             : ARNC0AUTCG_typ ;                  (* Compensation gear *)
   cam_prof             : ARNC0AUTCP_typ ;                  (* Cam profile *)
   event                : ARRAY [0..5] OF ARNC0AUTER_typ ;  (* Event *)
END_STRUCT;
ARNC0AUTOM_typ : STRUCT                                     (* Cam Profile Automat *)
   status               : ARNC0AUTST_typ ;                  (* Status *)
   signal1              : USINT ;                           (* Signal 1 from the PLC to the cam profile automat *)
   signal2              : USINT ;                           (* Signal 2 from the PLC to the cam profile automat *)
   signal3              : USINT ;                           (* Signal 3 from the PLC to the cam profile automat *)
   signal4              : USINT ;                           (* Signal 4 from the PLC to the cam profile automat *)
   init_stat            : ARNC0AUTID_typ ;                  (* INIT State (for INIT of a certain state) *)
   coupling             : ARNC0AUTCC_typ ;                  (* Coupling configuration *)
   global               : ARNC0AUTGL_typ ;                  (* Global Parameters *)
   basis                : ARNC0AUTBA_typ ;                  (* Basis state *)
   state                : ARRAY [0..5] OF ARNC0AUTSC_typ ;  (* State *)
END_STRUCT;
ARNC0AXCMPST_typ : STRUCT                                   (* Status *)
   init                 : USINT ;                           (* Initialized *)
   mode                 : USINT ;                           (* Mode *)
   reserve0             : UINT ;                            (* Reserved *)
END_STRUCT;
ARNC0AXCMPSSE_typ : STRUCT                                  (* Slope error compensation *)
   data_modul1          : ARRAY [0..11] OF USINT ;          (* Name of data module 1 *)
   data_modul2          : ARRAY [0..11] OF USINT ;          (* Name of data module 2 *)
   set_factor           : REAL ;                            (* Multiplication factor for set values *)
   corr_factor          : REAL ;                            (* Multiplication factor for corrected values *)
   start_offset         : REAL ;                            (* Start offset *)
END_STRUCT;
ARNC0AXCMPBL_typ : STRUCT                                   (* Backlash compensation *)
   s_init               : REAL ;                            (* Initial relative movement to mesh *)
   s                    : REAL ;                            (* Backlash *)
   v                    : REAL ;                            (* Velocity *)
   a                    : REAL ;                            (* Acceleration *)
END_STRUCT;
ARNC0AXCMPPA_typ : STRUCT                                   (* Compensation parameter *)
   mode                 : USINT ;                           (* Mode *)
   reserve0             : ARRAY [0..2] OF USINT ;           (* Reserved *)
   slope                : ARNC0AXCMPSSE_typ ;               (* Slope error compensation *)
   backlash             : ARNC0AXCMPBL_typ ;                (* Backlash compensation *)
END_STRUCT;
ARNC0AXCMP_typ : STRUCT                                     (* Axis Compensation *)
   status               : ARNC0AXCMPST_typ ;                (* Status *)
   parameter            : ARNC0AXCMPPA_typ ;                (* Parameters *)
END_STRUCT;
ARNC0AXMOV2_typ : STRUCT                                    (* Extended Axis movement *)
   cam_prof             : ARNC0CAMPR_typ ;                  (* Cam profile *)
   automat              : ARNC0AUTOM_typ ;                  (* Cam profile automat *)
   compensation         : ARNC0AXCMP_typ ;                  (* Compensation of axis errors *)
END_STRUCT;
ARNC0AXMOS_typ : STRUCT                                     (* Status Bits *)
   ds_warning           : USINT ;                           (* Lag error greater than "limit.ds_warning" *)
   reserve              : ARRAY [0..2] OF USINT ;           (* Reserved *)
END_STRUCT;
ARNC0AXMON_typ : STRUCT                                     (* Axis monitor *)
   s_act                : DINT ;                            (* Actual position *)
   s_set                : DINT ;                            (* Set position *)
   s_set_comp           : REAL ;                            (* Compensated set position *)
   v_set                : REAL ;                            (* Set speed *)
   v_set_comp           : REAL ;                            (* Compensated set speed *)
   status               : ARNC0AXMOS_typ ;                  (* Status bits *)
   reserve0             : ARRAY [0..2] OF UDINT ;           (* Reserved *)
END_STRUCT;
ARNC0MSSTA_typ : STRUCT                                     (* Status *)
   err_cl0              : USINT ;                           (* Error class 0 *)
   NOT_USE_1            : ARRAY [0..2] OF USINT ;
END_STRUCT;
ARNC0MSCNT_typ : STRUCT                                     (* Number of not acknowledged messages *)
   error                : UINT ;                            (* Count of not acknowledged errors *)
   NOT_USE_1            : ARRAY [0..5] OF USINT ;
END_STRUCT;
ARNC0MSREC_typ : STRUCT                                     (* Current message record *)
   number               : UDINT ;                           (* Number *)
   info                 : ARRAY [0..11] OF USINT ;          (* Additional Info *)
   NOT_USE_1            : ARRAY [0..1] OF USINT ;
   errorclass           : UINT ;                            (* Error class *)
   reserve              : UDINT ;                           (* Reserved *)
END_STRUCT;
ARNC0MTXST_typ : STRUCT                                     (* Status of text determination *)
   lines                : UINT ;                            (* Lines of the determined text *)
   error                : UINT ;                            (* Error *)
END_STRUCT;
ARNC0MTXPA_typ : STRUCT                                     (* Parameters for text determination *)
   format               : UINT ;                            (* Format *)
   columns              : UINT ;                            (* Number of columns per line *)
   data_modul           : ARRAY [0..11] OF USINT ;          (* Name of the data module *)
   data_len             : UINT ;                            (* Length of data buffer in application program *)
   reserve              : UINT ;                            (* Reserved *)
   data_adr             : UDINT ;                           (* Address of data buffer in application program *)
END_STRUCT;
ARNC0MSTXT_typ : STRUCT                                     (* Text determination for current message record *)
   status               : ARNC0MTXST_typ ;                  (* Status *)
   parameter            : ARNC0MTXPA_typ ;                  (* Parameters *)
END_STRUCT;
ARNC0MSG_typ : STRUCT                                       (* Messages *)
   status               : ARNC0MSSTA_typ ;                  (* Status *)
   count                : ARNC0MSCNT_typ ;                  (* Count of not acknowledged messages *)
   record               : ARNC0MSREC_typ ;                  (* Current message record *)
   text                 : ARNC0MSTXT_typ ;                  (* Text determination for current message record *)
END_STRUCT;
ARNC0NCTST_typ : STRUCT                                     (* NC Test *)
   Open_UseApplNcObj    : USINT ;                           (* Open test: Use the same NC object as the application *)
   Close_NoMoveAbort    : USINT ;                           (* Close test: No move abortion *)
   reserve1             : USINT ;                           (* Reserved *)
   reserve2             : USINT ;                           (* Reserved *)
END_STRUCT;
ARNC0AXIS_typ : STRUCT                                      (* ARNC0 - Axis *)
   NOT_USE_1            : ARRAY [0..5] OF USINT ;
   size                 : UINT ;                            (* Size of the corresponding NC manager data type *)
   sw_version           : ARNC0SWVER_typ ;                  (* Software Version ID *)
   nc_obj_inf           : ARNC0OBINF_typ ;                  (* NC Object Information *)
   simulation           : ARNC0AXSIM_typ ;                  (* Simulation Mode *)
   global               : ARNC0GLINI_typ ;                  (* Global Parameters *)
   network              : ARNC0NETAX_typ ;                  (* Network *)
   datblock             : ARNC0AXDBL_typ ;                  (* Data block operation *)
   dig_in               : ARNC0DIGIN_typ ;                  (* Digital Inputs *)
   encoder_if           : ARNC0ENCIF_typ ;                  (* Encoder Interface *)
   limit                : ARNC0AXLIM_typ ;                  (* Limit value *)
   controller           : ARNC0CTRL_typ ;                   (* Controller *)
   move                 : ARNC0AXMOV_typ ;                  (* Axis movement *)
   setup                : ARNC0SETUP_typ ;                  (* Setup *)
   NOT_USE_2            : ARRAY [0..119] OF USINT ;
   PLCopen_MC           : ARNC0PLCOPENAX_typ ;              (* PLCopen for Motion Components *)
   pos_latch            : ARNC0POS_L_typ ;                  (* Positioning latch *)
   move2                : ARNC0AXMOV2_typ ;                 (* Extended axis movement *)
   monitor              : ARNC0AXMON_typ ;                  (* Monitor *)
   message              : ARNC0MSG_typ ;                    (* Messages (errors, warnings) *)
   nc_test              : ARNC0NCTST_typ ;                  (* NC Test *)
   NOT_USE_3            : ARRAY [0..47] OF USINT ;
END_STRUCT;
ARNC0CNCSIM_typ : STRUCT                                    (* Simulation mode *)
   status               : USINT ;                           (* Status *)
   reserve              : ARRAY [0..2] OF USINT ;           (* Reserved *)
END_STRUCT;
ARNC0ACCADEX_typ : STRUCT                                   (* Reference Address *)
   access_adr           : UDINT ;                           (* Address for "access" *)
END_STRUCT;
ARNC0NCLIM_typ : STRUCT                                     (* CNC limits *)
   init                 : USINT ;                           (* Initialization complete *)
   reserve              : ARRAY [0..2] OF USINT ;           (* Reserved *)
   v                    : REAL ;                            (* Velocity *)
   a_pos                : REAL ;                            (* Positive acceleration *)
   a_neg                : REAL ;                            (* Negative acceleration *)
   t_jolt               : REAL ;                            (* Jolt time *)
   blocktransition      : USINT ;                           (* Mode for block transitions *)
   reserve0             : ARRAY [0..2] OF USINT ;           (* Reserved *)
   v_jump               : REAL ;                            (* Speed jump *)
   a_jump               : REAL ;                            (* Acceleration jump *)
   v_jump_t             : REAL ;                            (* Speed jump for tangential axis *)
   s_jump_t             : REAL ;                            (* Tangential deviation for subsequent path elements *)
   s_sync1_t            : UINT ;                            (* Synchrone M-Function at end of path element *)
   s_sync2_t            : UINT ;                            (* Synchrone M-Function at beginn of path element *)
   radius_err           : REAL ;                            (* Error of radius *)
   block_buffer         : UDINT ;                           (* Block buffer for backtracing the CNC path *)
   elements             : UINT ;                            (* Calculated elements before starting *)
   lookahead            : UINT ;                            (* Size of lookahead buffer *)
   halt                 : USINT ;                           (* Stop at passing beyond the submission values *)
   reserve1             : ARRAY [0..2] OF USINT ;           (* Reserved *)
   filter_err           : REAL ;                            (* Maximum contour error caused by "axis[i],t_axfilter" *)
   filter_err_trans     : REAL ;                            (* Maximum contour error at block transition caused by "axis[i],t_axfilter" *)
   plot                 : ARNC0ACCADEX_typ ;                (* Plot buffer *)
   dynamic              : ARNC0ACCADEX_typ ;                (* Dynamic buffer *)
END_STRUCT;
ARNC0SKPLM_typ : STRUCT                                     (* Interpreter skip level *)
   level_0              : USINT ;                           (* Skip level 0 *)
   level_1              : USINT ;                           (* Skip level 1 *)
   level_2              : USINT ;                           (* Skip level 2 *)
   level_3              : USINT ;                           (* Skip level 3 *)
   level_4              : USINT ;                           (* Skip level 4 *)
   level_5              : USINT ;                           (* Skip level 5 *)
   level_6              : USINT ;                           (* Skip level 6 *)
   level_7              : USINT ;                           (* Skip level 7 *)
   level_8              : USINT ;                           (* Skip level 8 *)
   level_9              : USINT ;                           (* Skip level 9 *)
   reserve0             : ARRAY [0..1] OF USINT ;           (* Reserved *)
END_STRUCT;
ARNC0NCMST_typ : STRUCT                                     (* Status CNC movement *)
   cnt_ncprog           : UINT ;                            (* Number of started CNC programs/blocks *)
   halt                 : USINT ;                           (* State "halt" *)
   halt_info            : USINT ;                           (* INFO aboute cause of "Halt" state *)
   m1_stop              : USINT ;                           (* Operating mode "Stop at M1" *)
   single_s             : USINT ;                           (* Operating mode "Single step" *)
   skip_fcn             : USINT ;                           (* Operating mode "Skip Function" *)
   dpr_ovr              : USINT ;                           (* "normal" override \  DPR-override *)
   skip_level           : ARNC0SKPLM_typ ;                  (* Skip level *)
END_STRUCT;
ARNC0NCSTO_typ : STRUCT                                     (* Stop Movement *)
   decel_ramp           : USINT ;                           (* Deceleration ramp *)
   reserve0             : USINT ;                           (* Reserved *)
   reserve1             : UINT ;                            (* Reserved *)
END_STRUCT;
ARNC0NCESTO_typ : STRUCT                                    (* Emergency Stop *)
   path                 : USINT ;                           (* Path behaviour *)
   reserve0             : USINT ;                           (* Reserved *)
   reserve1             : UINT ;                            (* Reserved *)
END_STRUCT;
ARNC0NCPRG_typ : STRUCT                                     (* CNC program *)
   name                 : ARRAY [0..99] OF USINT ;          (* Name of the NC data module *)
   init_prg             : ARRAY [0..99] OF USINT ;          (* Name of initial CNC program *)
   start_pos_type       : USINT ;                           (* Type of start position *)
   start_mode           : USINT ;                           (* Start mode for CNC program *)
   NOT_USE_1            : USINT ;
   delete_mode          : USINT ;                           (* Mode for deleting a CNC program *)
   start_pos            : DINT ;                            (* Starting position *)
   restart_type         : USINT ;                           (* Type of restart point *)
   reserve1             : ARRAY [0..2] OF USINT ;           (* Reserved *)
   block_ncprog         : UDINT ;                           (* Block number in CNC program *)
   offset_ncprog        : UDINT ;                           (* Offset (Byte) in current CNC program *)
   s_ncprog             : REAL ;                            (* Path position in current CNC program *)
   s_start              : ARRAY [0..14] OF REAL ;           (* Starting position *)
END_STRUCT;
ARNC0ACCAD_typ : STRUCT                                     (* Address for evaluation with "access" *)
   access_adr           : UDINT ;                           (* Address for "access" *)
END_STRUCT;
ARNC0SSTEP_typ : STRUCT                                     (* Single step *)
   mode                 : USINT ;                           (* Mode *)
   reserve0             : ARRAY [0..2] OF USINT ;           (* Reserved *)
   bit_pattern          : UDINT ;                           (* Bit pattern *)
END_STRUCT;
ARNC0SKPL_typ : STRUCT                                      (* Interpreter skip level *)
   level_0              : USINT ;                           (* Skip level 0 *)
   level_1              : USINT ;                           (* Skip level 1 *)
   level_2              : USINT ;                           (* Skip level 2 *)
   level_3              : USINT ;                           (* Skip level 3 *)
   level_4              : USINT ;                           (* Skip level 4 *)
   level_5              : USINT ;                           (* Skip level 5 *)
   level_6              : USINT ;                           (* Skip level 6 *)
   level_7              : USINT ;                           (* Skip level 7 *)
   level_8              : USINT ;                           (* Skip level 8 *)
   level_9              : USINT ;                           (* Skip level 9 *)
   reserve0             : ARRAY [0..1] OF USINT ;           (* Reserved *)
END_STRUCT;
ARNC0NCMOV_typ : STRUCT                                     (* CNC movement *)
   status               : ARNC0NCMST_typ ;                  (* Status *)
   stop                 : ARNC0NCSTO_typ ;                  (* Stop Movement *)
   e_stop               : ARNC0NCESTO_typ ;                 (* Emergency stop *)
   override             : INT ;                             (* Override *)
   R_override           : UINT ;                            (* Rapid override affects CNC path *)
   F_override           : UDINT ;                           (* Feedrate override affects CNC path *)
   ncprogram            : ARNC0NCPRG_typ ;                  (* NC program *)
   ncblock              : ARRAY [0..51] OF USINT ;          (* NC block *)
   dpr_ovr              : ARNC0ACCAD_typ ;                  (* "normal" override \  DPR-override *)
   dpr_if               : ARNC0ACCAD_typ ;                  (* DPR-interface *)
   single_s             : ARNC0SSTEP_typ ;                  (* Operating mode "Single step" *)
   skip_level           : ARNC0SKPL_typ ;                   (* Skip level *)
END_STRUCT;
ARNC0NCDST_typ : STRUCT                                     (* CNC decoder status *)
   halt                 : USINT ;                           (* State "halt" *)
   sync                 : USINT ;                           (* State "Waiting for SYNC" *)
   breakpt_halt         : USINT ;                           (* State "Halt at breakpoint" *)
   single_s_halt        : USINT ;                           (* State "Halt in single step mode" *)
   single_s             : UINT ;                            (* Operating mode "Single step" *)
   reserve              : UINT ;                            (* Reserved *)
   program_load         : UINT ;                            (* Status of 'program load' *)
   program_unload       : UINT ;                            (* Status of 'program unload' *)
   mp_log               : USINT ;                           (* Motion packet log *)
   reserve1             : ARRAY [0..2] OF USINT ;           (* Reserved *)
END_STRUCT;
ARNC0DCHLTINFO_typ : STRUCT                                 (* Interpreter halt info (e.g. breakpoint, single step) *)
   file_name            : ARRAY [0..99] OF USINT ;          (* File name *)
   program_name         : ARRAY [0..99] OF USINT ;          (* Program name *)
   subprog_name         : ARRAY [0..99] OF USINT ;          (* Sub program name *)
   line_nr              : UDINT ;                           (* Line number *)
   block_nr             : UDINT ;                           (* Block number *)
END_STRUCT;
ARNC0DCCDC_typ : STRUCT                                     (* Cutting Diameter Correction *)
   side                 : USINT ;                           (* Processing side Cutting Diameter Compensation *)
   entry                : USINT ;                           (* Select/deselect Cutting Diameter Compensation *)
   circ_transition      : USINT ;                           (* Insert Circular Transitions *)
   circ_replace         : USINT ;                           (* Replace arc with straight line *)
   contour_violation    : USINT ;                           (* Accept contour violations *)
   intersection_path    : USINT ;                           (* Additional intersection path calculation *)
   NOT_USE_1            : ARRAY [0..1] OF USINT ;
   feedrate             : UDINT ;                           (* Feedrate on Transition Circles *)
   v_path_contour       : USINT ;                           (* Feedrate affects CNC path *)
   exit                 : USINT ;                           (* Deselection Mode Cutting Diameter Compensation *)
   NOT_USE_2            : ARRAY [0..1] OF USINT ;
END_STRUCT;
ARNC0DCPAR_typ : STRUCT                                     (* CNC decoder parameter *)
   move_cmd             : USINT ;                           (* Movement command *)
   plane                : USINT ;                           (* Plane *)
   co_ords              : USINT ;                           (* Co-ordinate definition *)
   center               : USINT ;                           (* Center point definition *)
   v_path               : UDINT ;                           (* Path speed *)
   cdc                  : ARNC0DCCDC_typ ;                  (* Tool radius correction *)
   t_ax_period          : USINT ;                           (* Operating mode for  tangential axis *)
   system_unit          : USINT ;                           (* Measurement unit for CNC system *)
   v_path_mode          : USINT ;                           (* Mode for feed rate calculation *)
   reserve1             : USINT ;                           (* Reserved *)
   rot_pref_dir         : USINT ;                           (* Preferable direction of rotary axes *)
   limit_switch_mode    : USINT ;                           (* Mode for axis limit switch *)
   reserve0             : ARRAY [0..1] OF USINT ;           (* Reserved *)
END_STRUCT;
ARNC0DCDMO_typ : STRUCT                                     (* CNC decoder datamodule *)
   status               : ARNC0ACTST_typ ;                  (* Status *)
   zero_tab             : ARRAY [0..11] OF USINT ;          (* Data module name of zero point offset table *)
   tool_tab             : ARRAY [0..11] OF USINT ;          (* Data module name of tool data table *)
   rpar_tab             : ARRAY [0..11] OF USINT ;          (* Data module name of R parameter  table *)
END_STRUCT;
ARNC0R_PAR_typ : STRUCT                                     (* CNC decorder R-parameters *)
   status               : ARNC0ACTST_typ ;                  (* Status *)
   index                : UINT ;                            (* Index *)
   NOT_USE_1            : ARRAY [0..1] OF USINT ;
   value                : REAL ;                            (* R-Parameter-Value *)
END_STRUCT;
ARNC0DCSST_typ : STRUCT                                     (* Step mode debugger *)
   mode                 : UINT ;                            (* Mode *)
   number               : UINT ;                            (* Number of blocks to halt after *)
END_STRUCT;
ARNC0DCBRKPT_typ : STRUCT                                   (* Set Breakpoint *)
   file_name            : ARRAY [0..99] OF USINT ;          (* File name *)
   program_name         : ARRAY [0..99] OF USINT ;          (* Program name *)
   block_nr             : UDINT ;                           (* Block number *)
   line_nr              : UDINT ;                           (* Line number *)
END_STRUCT;
ARNC0DCBRKINFO_typ : STRUCT                                 (* Breakpoint info *)
   total_nr             : UDINT ;                           (* Total number of currently set breakpoints *)
   breakpoint_set       : ARRAY [0..4] OF ARNC0DCBRKPT_typ ;  (* Info to currently set breakpoints *)
END_STRUCT;
ARNC0DCBRKPAR_typ : STRUCT                                  (* Breakpoint Parameter *)
   file_name            : ARRAY [0..99] OF USINT ;          (* File name *)
   pos_type             : UDINT ;                           (* Type of break point *)
   position             : UDINT ;                           (* Block or line number *)
   break_count          : UDINT ;                           (* Halt on n’th hit *)
END_STRUCT;
ARNC0DCBRK_typ : STRUCT                                     (* Breakpoint *)
   status               : ARNC0ACTST_typ ;                  (* Status *)
   info                 : ARNC0DCBRKINFO_typ ;              (* INFO-function *)
   parameter            : ARNC0DCBRKPAR_typ ;               (* Parameters *)
END_STRUCT;
ARNC0DCEXPR_typ : STRUCT                                    (* Expression *)
   status               : ARNC0ACTST_typ ;                  (* Status *)
   query                : ARRAY [0..63] OF USINT ;          (* Variable/expression to evaluate *)
   result               : ARRAY [0..63] OF USINT ;          (* Result *)
END_STRUCT;
ARNC0DCVACCINFO_typ : STRUCT                                (* Info for access to variables *)
   address              : UDINT ;                           (* Access address to interpreter variable *)
   length               : UDINT ;                           (* Variable size (total number of byte) *)
   array_dim1           : UDINT ;                           (* First array dimension *)
   array_dim2           : UDINT ;                           (* Second array dimension *)
   data_type            : UINT ;                            (* Data type (see AS library “sys_lib”) *)
   scope                : UINT ;                            (* Variable scope *)
   synch_type           : UINT ;                            (* Synchronization type *)
   reserve0             : UINT ;                            (* Reserved *)
END_STRUCT;
ARNC0RVARACC_typ : STRUCT                                   (* Access to variables *)
   status               : ARNC0ACTST_typ ;                  (* Status *)
   name                 : ARRAY [0..31] OF USINT ;          (* Name of variable *)
   info                 : ARNC0DCVACCINFO_typ ;             (* INFO-function *)
END_STRUCT;
ARNC0NCDEC_typ : STRUCT                                     (* CNC decoder *)
   init                 : USINT ;                           (* Initialization complete *)
   reserve              : ARRAY [0..2] OF USINT ;           (* Reserved *)
   status               : ARNC0NCDST_typ ;                  (* Status *)
   halt_info            : ARNC0DCHLTINFO_typ ;              (* INFO aboute cause of "Halt" state *)
   parameter            : ARNC0DCPAR_typ ;                  (* Parameters *)
   data_modul           : ARNC0DCDMO_typ ;                  (* Data Modules *)
   r_param              : ARNC0R_PAR_typ ;                  (* R-parameter *)
   s_step               : ARNC0DCSST_typ ;                  (* Interpreter single step mode *)
   breakpoint           : ARNC0DCBRK_typ ;                  (* Breakpoints in CNC program *)
   expression           : ARNC0DCEXPR_typ ;                 (* Variable/Expression watch and force function *)
   var_access           : ARNC0RVARACC_typ ;                (* Direct access to Interpreter Variables *)
END_STRUCT;
ARNC0NCAXST_typ : STRUCT                                    (* Status *)
   add_par_id           : UINT ;                            (* Parameter ID of the additive element for the cyclic set position *)
   reserve              : ARRAY [0..1] OF USINT ;           (* Reserved *)
END_STRUCT;
ARNC0TRC_typ : STRUCT                                       (* Trigger Configuration *)
   trigger1_pos         : USINT ;                           (* Trigger1: Positive edge *)
   trigger1_neg         : USINT ;                           (* Trigger1: Negative edge *)
   trigger2_pos         : USINT ;                           (* Trigger2: Positive edge *)
   trigger2_neg         : USINT ;                           (* Trigger2: Negative edge *)
END_STRUCT;
ARNC0NCTRG_typ : STRUCT                                     (* Source for Hardware Trigger *)
   nc_object            : UDINT ;                           (* NC object or ncOFF *)
   nc_object_plcopen    : UDINT ;                           (* NC object or ncOFF *)
   NOT_USE_1            : ARRAY [0..3] OF USINT ;
   trg_conf             : ARNC0TRC_typ ;                    (* Trigger Configuration *)
END_STRUCT;
ARNC0NCAXSSE_typ : STRUCT                                   (* Axes error compensation *)
   active               : USINT ;                           (* Active *)
   reserve              : ARRAY [0..2] OF USINT ;           (* Reserved *)
   cmp_data             : ARNC0ACCADEX_typ ;                (* Compensation data *)
END_STRUCT;
ARNC0NCAXP_typ : STRUCT                                     (* CNC-axis settings *)
   NOT_USE_1            : ARRAY [0..71] OF USINT ;
   status               : ARNC0NCAXST_typ ;                 (* Status *)
   nc_object            : UDINT ;                           (* NC object or ncOFF *)
   nc_object_plcopen    : UDINT ;                           (* NC object or ncOFF *)
   name                 : ARRAY [0..13] OF USINT ;          (* Name of the axis in the CNC program *)
   reserve3             : ARRAY [0..1] OF USINT ;           (* Reserved *)
   type                 : UDINT ;                           (* Type *)
   ipl_mode             : USINT ;                           (* Interpolation mode *)
   reserve4             : ARRAY [0..2] OF USINT ;           (* Reserved *)
   unitfactor           : REAL ;                            (* Multiplication factor of the units *)
   t_axfilter           : REAL ;                            (* Filter time for axis jolt filter *)
   drive_axfilter       : USINT ;                           (* Axis jolt filter on the drive during CNC movement *)
   reserve2             : ARRAY [0..2] OF USINT ;           (* Reserved *)
   rot_period           : REAL ;                            (* Period of rotary axis *)
   rot_offset           : REAL ;                            (* Start of period for rotary axis *)
   add_par_id           : UINT ;                            (* Parameter ID of the additive element for the cyclic set position *)
   reserve5             : ARRAY [0..1] OF USINT ;           (* Reserved *)
   trg_source           : ARNC0NCTRG_typ ;                  (* Trigger Source *)
   ax_compensation      : ARNC0NCAXSSE_typ ;                (* Axis error compensatioin *)
END_STRUCT;
ARNC0NCEXAXP_typ : STRUCT                                   (* External CNC axis parameters *)
   nc_object            : ARRAY [0..14] OF UDINT ;          (* NC object or ncOFF *)
END_STRUCT;
ARNC0NCAXCMP_typ : STRUCT                                   (* Compensation parameter for Cartesian axes *)
   matrix_el            : ARRAY [0..8] OF REAL ;            (* Element of compensation matrix *)
END_STRUCT;
ARNC0NCAXTRF_typ : STRUCT                                   (* Kinematic transformation parameters *)
   name                 : ARRAY [0..99] OF USINT ;          (* Name of the NC data module *)
   trf_full             : USINT ;                           (* Full kinematic transformation *)
   trf_type             : USINT ;                           (* Type of kinematic transformation *)
   reserve0             : ARRAY [0..1] OF USINT ;           (* Reserved *)
   axes_tcp             : ARRAY [0..11] OF USINT ;          (* Index of path axes *)
   axes_joint           : ARRAY [0..11] OF USINT ;          (* Index of joint axes *)
   axes_frame           : ARRAY [0..5] OF USINT ;           (* Index of frame axis [dx, dy, dz, phi, theta, psi] *)
   reserve1             : ARRAY [0..1] OF USINT ;           (* Reserved *)
   tcp_add_el           : ARRAY [0..11] OF REAL ;           (* Additive element of path axes *)
   joint_add_el         : ARRAY [0..11] OF REAL ;           (* Additive element of joint axes *)
   frame_add_el         : ARRAY [0..5] OF REAL ;            (* Additive element of frame axes *)
   d_full_add_el        : ARRAY [0..5] OF REAL ;            (* Additive element of general tools (D_FULL) *)
   in_pos_tolerance     : REAL ;                            (* Position tolerance for path axes at beginning of a movement *)
END_STRUCT;
ARNC0AXP_ARR_typ : STRUCT                                   (* Datatype for the AXP-array *)
   init                 : USINT ;                           (* Initialization complete *)
   reserve              : ARRAY [0..2] OF USINT ;           (* Reserved *)
   axis                 : ARRAY [0..14] OF ARNC0NCAXP_typ ;  (* NC axis *)
   ext_ax_parameter     : ARNC0NCEXAXP_typ ;                (* External CNC axis parameters *)
   compensation         : ARNC0NCAXCMP_typ ;                (* Compensation parameter for Cartesian axes *)
   transformation       : ARNC0NCAXTRF_typ ;                (* Kinematic Transformation *)
END_STRUCT;
ARNC0PLCPA_typ : STRUCT                                     (* CNC-PLC parameters *)
   t_fcn_init           : USINT ;                           (* Initialize T function with CNC-Reset *)
   s_fcn_init           : USINT ;                           (* Initialize S function with CNC-Reset *)
   first_M              : UINT ;                            (* Index of first M function without synchronization *)
   last_M               : UINT ;                            (* Index of last M function without synchronization *)
   first_M_S            : UINT ;                            (* Index of first M function with synchronization *)
   last_M_S             : UINT ;                            (* Index of last M function with synchronization *)
   NOT_USE_1            : ARRAY [0..1] OF USINT ;
END_STRUCT;
ARNC0PLCDA_typ : STRUCT                                     (* CNC-PLC data *)
   t_funct              : UINT ;                            (* T function value *)
   NOT_USE_1            : ARRAY [0..1] OF USINT ;
   s_funct              : ARRAY [0..3] OF UDINT ;           (* S function values *)
   m_funct              : ARRAY [0..1023] OF USINT ;        (* Display for "Execute M Function" *)
END_STRUCT;
ARNC0EXP_typ : STRUCT                                       (* External CNC-PLC parameters *)
   status               : USINT ;                           (* Status *)
   reserve              : ARRAY [0..2] OF USINT ;           (* Reserved *)
   access_adr           : UDINT ;                           (* Address for "access" *)
END_STRUCT;
ARNC0NCPLC_typ : STRUCT                                     (* CNC-PLC data *)
   init                 : USINT ;                           (* Initialization complete *)
   reserve              : ARRAY [0..2] OF USINT ;           (* Reserved *)
   parameter            : ARNC0PLCPA_typ ;                  (* Parameters *)
   data                 : ARNC0PLCDA_typ ;                  (* Data *)
   ex_param             : ARNC0EXP_typ ;                    (* External parameter *)
   m_param              : ARNC0ACCAD_typ ;                  (* M parameters *)
END_STRUCT;
ARNC0ENST_typ : STRUCT                                      (* Status *)
   enabled              : USINT ;                           (* Enabled *)
   active               : USINT ;                           (* Active *)
   data_valid           : USINT ;                           (* Valid restart data available *)
   data_saved           : USINT ;                           (* Restart data saved (since last program start) *)
END_STRUCT;
ARNC0NCRSR_typ : STRUCT                                     (* Result *)
   name                 : ARRAY [0..99] OF USINT ;          (* Name of the NC data module *)
   init_prg             : ARRAY [0..99] OF USINT ;          (* Name of initial CNC program *)
   start_pos_type       : USINT ;                           (* Type of start position *)
   start_mode           : USINT ;                           (* Start mode for CNC program *)
   reserve              : UINT ;                            (* Reserved *)
   start_pos            : DINT ;                            (* Starting position *)
   restart_type         : USINT ;                           (* Type of restart point *)
   reserve1             : ARRAY [0..2] OF USINT ;           (* Reserved *)
   block_ncprog         : UDINT ;                           (* Block number in CNC program *)
   offset_ncprog        : UDINT ;                           (* Offset (Byte) in current CNC program *)
   line_ncprog          : UDINT ;                           (* Line number in CNC program *)
   s_ncprog             : REAL ;                            (* Path position in current CNC program *)
   s_set                : ARRAY [0..14] OF REAL ;           (* Set position *)
END_STRUCT;
ARNC0NCRSP_typ : STRUCT                                     (* Parameter *)
   restart_type         : USINT ;                           (* Type of restart point *)
   NOT_USE_1            : ARRAY [0..2] OF USINT ;
   block_ncprog         : UDINT ;                           (* Block number in CNC program *)
   offset_ncprog        : UDINT ;                           (* Offset (Byte) in current CNC program *)
   s_ncprog             : REAL ;                            (* Path position in current CNC program *)
END_STRUCT;
ARNC0NCRSI_typ : STRUCT                                     (* INFO-function *)
   status               : ARNC0ACTST_typ ;                  (* Status *)
   result               : ARNC0NCRSR_typ ;                  (* Result *)
   parameter            : ARNC0NCRSP_typ ;                  (* Parameters *)
END_STRUCT;
ARNC0NCRPA_typ : STRUCT                                     (* General restart parameters *)
   param_buffer         : UDINT ;                           (* Buffer size for R- and EX- parameters *)
   trigger_buffer       : UDINT ;                           (* Buffer size for trigger blocks *)
END_STRUCT;
ARNC0NCRST_typ : STRUCT                                     (* Restart of a NC-program *)
   status               : ARNC0ENST_typ ;                   (* Status *)
   info                 : ARNC0NCRSI_typ ;                  (* INFO-function *)
   parameter            : ARNC0NCRPA_typ ;                  (* Parameters *)
END_STRUCT;
ARNC0RDMOD_typ : STRUCT                                     (* Datamodule handling *)
   status               : ARNC0ACTST_typ ;                  (* Status *)
   name                 : ARRAY [0..11] OF USINT ;          (* Name of the NC data module *)
END_STRUCT;
ARNC0NCMNPAR_typ : STRUCT                                   (* CNC monitor parameter *)
   pos_mode             : USINT ;                           (* CNC Position monitor *)
   block_mode           : USINT ;                           (* Blocks display mode *)
   line_nr_mode         : USINT ;                           (* Display line numbers *)
   max_call_level       : USINT ;                           (* Max. call level for extended block numbers *)
   access_adr           : UDINT ;                           (* Address for "access" *)
END_STRUCT;
ARNC0NCMNS_typ : STRUCT                                     (* CNC monitor status *)
   zeropoff             : USINT ;                           (* Mode "Subtract zero point offset from positions" *)
   pos_mode             : USINT ;                           (* CNC Position monitor *)
   NOT_USE_1            : USINT ;
   block_mode           : USINT ;                           (* Blocks display mode *)
   line_nr_mode         : USINT ;                           (* Display line numbers *)
   s_set_valid          : USINT ;                           (* Set positions valid in the CNC monitor *)
   NOT_USE_2            : ARRAY [0..1] OF USINT ;
END_STRUCT;
ARNC0NCMON_typ : STRUCT                                     (* CNC monitor *)
   parameter            : ARNC0NCMNPAR_typ ;                (* Parameters *)
   status               : ARNC0NCMNS_typ ;                  (* Status *)
   s_set                : ARRAY [0..14] OF REAL ;           (* Set position *)
   s_ncblock            : ARRAY [0..14] OF REAL ;           (* Axis distance until end of current NC block *)
   v_path               : REAL ;                            (* Path speed *)
   nr_ncprog            : UDINT ;                           (* Number of current CNC program *)
   name_ncprog          : ARRAY [0..99] OF USINT ;          (* Name of current CNC program *)
   pos_ncprog           : UDINT ;                           (* Position in current CNC program *)
   block_ncprog         : UDINT ;                           (* Block number in CNC program *)
   line_ncprog          : UDINT ;                           (* Line number in CNC program *)
   call_level           : USINT ;                           (* Current call level for sub-programs *)
   reserve1             : ARRAY [0..2] OF USINT ;           (* Reserved *)
   t_ncprog             : REAL ;                            (* Run-Time of current CNC program *)
   s_ncprog             : REAL ;                            (* Path position in current CNC program *)
   v_ncprog             : REAL ;                            (* Path speed currently defined in CNC program *)
   d_full               : ARRAY [0..5] OF REAL ;            (* Active D_FULL data *)
   tool_nr              : UINT ;                            (* Number of active tool data record *)
   zero_idx             : UINT ;                            (* Index of active absolute zero point offset *)
   type_ncblock         : UINT ;                            (* Type of current NC block *)
   PSM_phase            : UINT ;                            (* Path speed mode, phase *)
   t_dwell              : REAL ;                            (* Remaining time for G04 (dwell) *)
   ncblocks             : ARNC0ACCAD_typ ;                  (* Display of CNC blocks *)
   c_transform          : ARNC0ACCAD_typ ;                  (* Transformation matrices for coordinate systems *)
   ip_monitor           : ARNC0ACCAD_typ ;                  (* Interpreter monitor *)
   ext_monitor          : ARNC0ACCAD_typ ;                  (* Extended CNC Monitor *)
END_STRUCT;
ARNC0ERRCL0_typ : STRUCT                                    (* Error class 0 *)
   number               : ARRAY [0..19] OF UDINT ;          (* Number *)
END_STRUCT;
ARNC0CNC_typ : STRUCT                                       (* ARNC0 - CNC-System *)
   NOT_USE_1            : ARRAY [0..3] OF USINT ;
   size                 : UINT ;                            (* Size of the corresponding NC manager data type *)
   reserve0             : UINT ;                            (* Reserved *)
   sw_version           : ARNC0SWVER_typ ;                  (* Software Version ID *)
   nc_obj_inf           : ARNC0OBINF_typ ;                  (* NC Object Information *)
   simulation           : ARNC0CNCSIM_typ ;                 (* Simulation Mode *)
   global               : ARNC0GLINI_typ ;                  (* Global Parameters *)
   limit                : ARNC0NCLIM_typ ;                  (* Limit value *)
   move                 : ARNC0NCMOV_typ ;                  (* Movement *)
   decoder              : ARNC0NCDEC_typ ;                  (* Decoder *)
   axis                 : ARNC0AXP_ARR_typ ;                (* NC axis *)
   cnc_plc              : ARNC0NCPLC_typ ;                  (* CNC-PLC-Data *)
   restart              : ARNC0NCRST_typ ;                  (* RESTART of a CNC program *)
   data_modul           : ARNC0RDMOD_typ ;                  (* Data Modules *)
   monitor              : ARNC0NCMON_typ ;                  (* Monitor *)
   message              : ARNC0MSG_typ ;                    (* Messages (errors, warnings) *)
   err_cl0              : ARNC0ERRCL0_typ ;                 (* Error class 0 *)
   NOT_USE_2            : ARRAY [0..7] OF USINT ;
   nc_test              : ARNC0NCTST_typ ;                  (* NC Test *)
   NOT_USE_3            : ARRAY [0..47] OF USINT ;
END_STRUCT;
ARNC0EXPAR_typ : STRUCT                                     (* External CNC parameters *)
   EXB                  : ARRAY [0..99] OF SINT ;           (* EX(ternal) B(yte)-Parameters *)
   EXW                  : ARRAY [0..99] OF INT ;            (* EX(terne) W(ord)-Parameters *)
   EXL                  : ARRAY [0..99] OF DINT ;           (* EX(terne) L(ong)-Parameters *)
   EXF                  : ARRAY [0..99] OF REAL ;           (* EX(terne) F(loat)-Parameters *)
END_STRUCT;
ARNC0EXESL_typ : STRUCT                                     (* Scaling for the load *)
   units                : UDINT ;                           (* Units at the load *)
   rev_encod            : UDINT ;                           (* Encoder revolutions *)
END_STRUCT;
ARNC0EXESC_typ : STRUCT                                     (* Scaling for encoder interface *)
   load                 : ARNC0EXESL_typ ;                  (* Load *)
END_STRUCT;
ARNC0EXEPA_typ : STRUCT                                     (* Parameters for encoder interface *)
   count_dir            : USINT ;                           (* Count direction *)
   NOT_USE_1            : ARRAY [0..2] OF USINT ;
   scaling              : ARNC0EXESC_typ ;                  (* Scaling *)
END_STRUCT;
ARNC0EXEIF_typ : STRUCT                                     (* Encoder interface *)
   init                 : USINT ;                           (* Encoder interface initialized *)
   NOT_USE_1            : ARRAY [0..2] OF USINT ;
   parameter            : ARNC0EXEPA_typ ;                  (* Parameters *)
END_STRUCT;
ARNC0EXENW_typ : STRUCT                                     (* Network *)
   phase                : USINT ;                           (* Phase *)
   init                 : USINT ;                           (* Network initialized *)
   NOT_USE_1            : ARRAY [0..1] OF USINT ;
END_STRUCT;
ARNC0EXEHST_typ : STRUCT                                    (* Homing Status *)
   ok                   : USINT ;                           (* Reference position valid *)
   NOT_USE_1            : ARRAY [0..2] OF USINT ;
END_STRUCT;
ARNC0EXEHPA_typ : STRUCT                                    (* Homing Parameter *)
   s                    : DINT ;                            (* Reference position *)
   ref_pulse            : USINT ;                           (* Reference pulse *)
   NOT_USE_1            : ARRAY [0..2] OF USINT ;
END_STRUCT;
ARNC0EXEHOM_typ : STRUCT                                    (* Homing *)
   init                 : USINT ;                           (* Homing procedure initialized *)
   NOT_USE_1            : ARRAY [0..2] OF USINT ;
   status               : ARNC0EXEHST_typ ;                 (* Status *)
   parameter            : ARNC0EXEHPA_typ ;                 (* Parameters *)
END_STRUCT;
ARNC0EXEMOV_typ : STRUCT                                    (* Movement *)
   homing               : ARNC0EXEHOM_typ ;                 (* Homing procedure *)
END_STRUCT;
ARNC0EXEPOS_typ : STRUCT                                    (* Filter for actual positions *)
   status               : USINT ;                           (* Status *)
   NOT_USE_1            : ARRAY [0..2] OF USINT ;
   t_filter             : REAL ;                            (* Filter time for extrapolation filter *)
   t_filter2            : REAL ;                            (* Filter time for disturbance filter *)
END_STRUCT;
ARNC0EXMON_typ : STRUCT                                     (* Monitor *)
   s_act                : DINT ;                            (* Actual position *)
   v_act                : REAL ;                            (* Actual speed *)
END_STRUCT;
ARNC0EXTEN_typ : STRUCT                                     (* ARNC0 - External Encoder *)
   NOT_USE_1            : ARRAY [0..3] OF USINT ;
   size                 : UINT ;                            (* Size of the corresponding NC manager data type *)
   NOT_USE_2            : ARRAY [0..1] OF USINT ;
   sw_version           : ARNC0SWVER_typ ;                  (* Software Version ID *)
   nc_obj_inf           : ARNC0OBINF_typ ;                  (* NC Object Information *)
   encoder_if           : ARNC0EXEIF_typ ;                  (* Encoder Interface *)
   network              : ARNC0EXENW_typ ;                  (* Network *)
   move                 : ARNC0EXEMOV_typ ;                 (* Movement *)
   act_pos              : ARNC0EXEPOS_typ ;                 (* Filter for actual position *)
   monitor              : ARNC0EXMON_typ ;                  (* Monitor *)
   message              : ARNC0MSG_typ ;                    (* Messages (errors, warnings) *)
   NOT_USE_3            : ARRAY [0..47] OF USINT ;
END_STRUCT;
ARNC0M_PAR_typ : STRUCT                                     (* CNC M parameters *)
   MW                   : ARRAY [0..99] OF INT ;            (* M-W(ord)-Parameters *)
   ML                   : ARRAY [0..99] OF DINT ;           (* M-L(ong)-Parameters *)
   MF                   : ARRAY [0..99] OF REAL ;           (* M-F(loat)-Parameters *)
END_STRUCT;
ARNC0INIST_typ : STRUCT                                     (* Status *)
   init                 : USINT ;                           (* Network initialized *)
   reserve              : ARRAY [0..2] OF USINT ;           (* Reserved *)
END_STRUCT;
ARNC0NETMO_typ : STRUCT                                     (* Network *)
   status               : ARNC0INIST_typ ;                  (* Status *)
END_STRUCT;
ARNC0DATMO_typ : STRUCT                                     (* Datamodule handling *)
   status               : ARNC0ACTST_typ ;                  (* Status *)
   NOT_USE_1            : USINT ;
   type                 : USINT ;                           (* Type *)
   reserve              : ARRAY [0..1] OF USINT ;           (* Reserved *)
   name                 : ARRAY [0..11] OF USINT ;          (* Name of the NC data module *)
END_STRUCT;
ARNC0TRTRI_typ : STRUCT                                     (* Trace trigger-point *)
   nc_object            : UDINT ;                           (* NC object or ncOFF *)
   type                 : USINT ;                           (* Type of the point *)
   event                : USINT ;                           (* Event *)
   NOT_USE_1            : ARRAY [0..1] OF USINT ;
   threshold            : REAL ;                            (* Threshold *)
END_STRUCT;
ARNC0TRTST_typ : STRUCT                                     (* Trace test-point *)
   nc_object            : UDINT ;                           (* NC object or ncOFF *)
   type                 : USINT ;                           (* Type of the point *)
   reserve              : ARRAY [0..2] OF USINT ;           (* Reserved *)
END_STRUCT;
ARNC0TRACE_typ : STRUCT                                     (* Trace *)
   status               : USINT ;                           (* Status *)
   reserve              : ARRAY [0..2] OF USINT ;           (* Reserved *)
   t_trace              : REAL ;                            (* Recording time *)
   t_sampling           : REAL ;                            (* Sampling time *)
   t_delay              : REAL ;                            (* Time of delay *)
   trigger              : ARNC0TRTRI_typ ;                  (* Trigger *)
   test_dat             : ARRAY [0..9] OF ARNC0TRTST_typ ;  (* Test data *)
   access_adr           : UDINT ;                           (* Address for "access" *)
END_STRUCT;
ARNC0MODUL_typ : STRUCT                                     (* For object-type ncMODUL *)
   NOT_USE_1            : ARRAY [0..3] OF USINT ;
   size                 : UINT ;                            (* Size of the corresponding NC manager data type *)
   reserve0             : UINT ;                            (* Reserved *)
   sw_version           : ARNC0SWVER_typ ;                  (* Software Version ID *)
   nc_obj_inf           : ARNC0OBINF_typ ;                  (* NC Object Information *)
   network              : ARNC0NETMO_typ ;                  (* Network *)
   data_modul           : ARNC0DATMO_typ ;                  (* Data Modules *)
   NOT_USE_2            : ARRAY [0..3] OF USINT ;
   message              : ARNC0MSG_typ ;                    (* Messages (errors, warnings) *)
   command              : ARNC0ACCAD_typ ;                  (* Command interface *)
   response             : ARNC0ACCAD_typ ;                  (* Response interface *)
   usertask             : ARNC0ACCAD_typ ;                  (* UserTask *)
   trace                : ARNC0TRACE_typ ;                  (* Trace *)
   NOT_USE_3            : ARRAY [0..51] OF USINT ;
END_STRUCT;
ARNC0NCCTR_typ : STRUCT                                     (* Transformations coordniate system *)
   handshake            : UINT ;                            (* Handshake *)
   NOT_USE_1            : ARRAY [0..1] OF USINT ;
   G92_matrix           : ARRAY [0..8] OF REAL ;            (* G92 matrix *)
   G192_matrix          : ARRAY [0..8] OF REAL ;            (* G192 matrix *)
   G292_matrix          : ARRAY [0..8] OF REAL ;            (* G292 matrix *)
   comp_matrix          : ARRAY [0..8] OF REAL ;            (* Compensation matrix *)
   offset               : ARRAY [0..14] OF REAL ;           (* Offset *)
END_STRUCT;
ARNC0NCDPR_typ : STRUCT                                     (* NC DPR *)
   halt_ncsz            : USINT ;                           (* Halt the CNC move at the end of an NC record *)
   halt                 : USINT ;                           (* Halt the CNC move *)
   NOT_USE_1            : ARRAY [0..1] OF USINT ;
END_STRUCT;
ARNC0NCSMO_typ : STRUCT                                     (* NC Monitor *)
   handshake            : UINT ;                            (* Handshake *)
   NOT_USE_1            : ARRAY [0..1] OF USINT ;
   ncblock_l2           : ARRAY [0..79] OF USINT ;          (* NC block *)
   ncblock_l1           : ARRAY [0..79] OF USINT ;          (* NC block *)
   ncblock              : ARRAY [0..79] OF USINT ;          (* NC block *)
   ncblock_n1           : ARRAY [0..79] OF USINT ;          (* NC block *)
   ncblock_n2           : ARRAY [0..79] OF USINT ;          (* NC block *)
   s_ncblock            : REAL ;                            (* Remaining path length until end of current NC block *)
   s_ncblock_tot        : REAL ;                            (* Path length of current NC block *)
   s_ncblock_n1         : REAL ;                            (* Path length of next NC block *)
END_STRUCT;
ARNC0PTRTR_typ : STRUCT                                     (* Trigger *)
   par_id               : UINT ;                            (* Parameter ID *)
   event                : USINT ;                           (* Event *)
   reserve              : USINT ;                           (* Reserved *)
   threshold            : REAL ;                            (* Threshold *)
   window               : REAL ;                            (* Latch window *)
END_STRUCT;
ARNC0PTRDA_typ : STRUCT                                     (* Test data *)
   par_id               : UINT ;                            (* Parameter ID *)
   reserve              : UINT ;                            (* Reserved *)
END_STRUCT;
ARNC0PTRSV_typ : STRUCT                                     (* Operating System Variable *)
   data_type            : USINT ;                           (* Data type *)
   reserve1             : USINT ;                           (* Reserved *)
   reserve2             : UINT ;                            (* Reserved *)
   address              : UDINT ;                           (* Address *)
END_STRUCT;
ARNC0PTRSY_typ : STRUCT                                     (* Configuration of Operating System Variables *)
   trigger              : ARNC0PTRSV_typ ;                  (* Trigger *)
   test_dat             : ARRAY [0..9] OF ARNC0PTRSV_typ ;  (* Test data *)
END_STRUCT;
ARNC0PATRC_typ : STRUCT                                     (* Trace *)
   status               : USINT ;                           (* Status *)
   reserve              : ARRAY [0..2] OF USINT ;           (* Reserved *)
   buf_size             : UDINT ;                           (* Size of trace data buffer on the drive *)
   NOT_USE_1            : ARRAY [0..3] OF USINT ;
   t_trace              : REAL ;                            (* Recording time *)
   t_sampling           : REAL ;                            (* Sampling time *)
   t_delay              : REAL ;                            (* Start delay *)
   trigger              : ARNC0PTRTR_typ ;                  (* Trigger *)
   test_dat             : ARRAY [0..9] OF ARNC0PTRDA_typ ;  (* Test data *)
   system_var           : ARNC0PTRSY_typ ;                  (* Configuration of Operating System Variables *)
END_STRUCT;
ARNC0PTRIN_typ : STRUCT                                     (* Internal for Parameter Trace *)
   errortext            : USINT ;                           (* Error text *)
   err_cl0              : USINT ;                           (* Error class 0 *)
   reserve              : UINT ;                            (* Reserved *)
END_STRUCT;
ARNC0PARTRACE_typ : STRUCT                                  (* ncPARID_TRACE-structure for ARNC0 *)
   NOT_USE_1            : ARRAY [0..3] OF USINT ;
   size                 : UINT ;                            (* Size of the corresponding NC manager data type *)
   reserve0             : UINT ;                            (* Reserved *)
   sw_version           : ARNC0SWVER_typ ;                  (* Software Version ID *)
   nc_obj_inf           : ARNC0OBINF_typ ;                  (* NC Object Information *)
   network              : ARNC0NETMO_typ ;                  (* Network *)
   trace                : ARNC0PATRC_typ ;                  (* Trace *)
   message              : ARNC0MSG_typ ;                    (* Messages (errors, warnings) *)
   intern               : ARNC0PTRIN_typ ;                  (* Intern *)
   NOT_USE_2            : ARRAY [0..47] OF USINT ;
END_STRUCT;
ARNC0MATRIX_typ : STRUCT                                    (* Rotation matrix *)
   matrix_el            : ARRAY [0..8] OF REAL ;            (* Element of compensation matrix *)
END_STRUCT;
ARNC0PLOTDATA_typ : STRUCT                                  (* Plot data in buffer *)
   block_ncprog         : UDINT ;                           (* Block number in CNC program *)
   cmd_code             : USINT ;                           (* Code of the command *)
   reserve0             : USINT ;                           (* Reserved *)
   info                 : USINT ;                           (* Additional Info *)
   plane                : USINT ;                           (* Plane *)
   end                  : ARRAY [0..2] OF REAL ;            (* End Point *)
   center               : ARRAY [0..2] OF REAL ;            (* Center point definition *)
   rotation             : ARNC0MATRIX_typ ;                 (* Rotation matrix *)
   v_ncprog             : REAL ;                            (* Path speed currently defined in CNC program *)
END_STRUCT;
ARNC0PLOTFOOTER_typ : STRUCT                                (* End of plot buffer *)
   buffer_end           : UDINT ;                           (* End of buffer *)
END_STRUCT;
ARNC0PLOTHEADER_typ : STRUCT                                (* Header for plot buffer *)
   size                 : UDINT ;                           (* Size of the corresponding NC manager data type *)
   format               : USINT ;                           (* Format *)
   status               : USINT ;                           (* Status *)
   reserve0             : UINT ;                            (* Reserved *)
   sw_version           : ARNC0SWVER_typ ;                  (* Software Version ID *)
   start                : UDINT ;                           (* Start *)
   write                : UDINT ;                           (* Reference for write access *)
   read                 : UDINT ;                           (* Reference for read access *)
END_STRUCT;
ARNC0DBLST_typ : STRUCT                                     (* Status *)
   data_len             : UDINT ;                           (* Length of data *)
   init                 : USINT ;                           (* Data block initialized *)
   ok                   : USINT ;                           (* Operation complete *)
   error                : USINT ;                           (* Error *)
   reserve1             : USINT ;                           (* Reserved *)
   reserve2             : UDINT ;                           (* Reserved *)
END_STRUCT;
ARNC0DBLPA_typ : STRUCT                                     (* Parameters *)
   data_len             : UDINT ;                           (* Length of data *)
   data_adr             : UDINT ;                           (* Data address *)
   data_modul           : ARRAY [0..11] OF USINT ;          (* Name of the data module *)
   index                : UINT ;                            (* Index *)
   mode                 : UINT ;                            (* Mode *)
   format               : UINT ;                            (* Format *)
   reserve              : UINT ;                            (* Reserved *)
END_STRUCT;
ARNC0DATBL_typ : STRUCT                                     (* Data block operation *)
   status               : ARNC0DBLST_typ ;                  (* Status *)
   parameter            : ARNC0DBLPA_typ ;                  (* Parameters *)
END_STRUCT;
ARNC0DNCHEADER_typ : STRUCT                                 (* Header of DNC Interface *)
   status               : USINT ;                           (* Status *)
   reserve              : ARRAY [0..2] OF USINT ;           (* Reserved *)
   start_adr            : UDINT ;                           (* Start address of CNC data area *)
   write_adr            : UDINT ;                           (* Write address (write pointer) *)
   read_adr             : UDINT ;                           (* Read address (read pointer) *)
   size                 : UDINT ;                           (* Size of CNC data area *)
END_STRUCT;
ARNC0TYPES_typ : STRUCT                                     (* Data structure for additional data types *)
   data_block           : ARNC0DATBL_typ ;                  (* Data block operation *)
   dnc_header           : ARNC0DNCHEADER_typ ;              (* Header of DNC Interface *)
END_STRUCT;
END_TYPE
```
